(* IEC 61131-3 sources: volt/packages/volt-lsp-iec/test-corpus/lenze-mid/Device/Plc Logic/Application/Library Manager/L_MC4P_RoboticHandling, 315 files *)

(* ---- IDENT_IN_GROUP_REF.dut ---- *)
TYPE IDENT_IN_GROUP_REF :
(
	NONE := 0,
	X := 1,
	Y := 2,
	Z := 3,
	A := 4,
	B := 5,
	C := 6,
	A1 := 7,
	A2 := 8,
	A3 := 9,
	A4 := 10,
	A5 := 11,
	A6 := 12,
	AUX1 := 13,
	AUX2 := 14,
	AUX3 := 15,
	AUX4 := 16,
	AUX5 := 17,
	AUX6 := 18
);
END_TYPE

(* ---- L_MC4P_AGBC_PARAMETER.dut ---- *)
TYPE L_MC4P_AGBC_PARAMETER :
STRUCT
	LRCARTESIANJOGVEL : LREAL := 10;
	LRCARTESIANJOGACC : LREAL := 100;
	LRCARTESIANJOGDEC : LREAL := 200;
	LRCARTESIANJOGJERK : LREAL := 10000;
	LRORIENTATIONJOGVEL : LREAL := 5;
	LRORIENTATIONJOGACC : LREAL := 50;
	LRORIENTATIONJOGDEC : LREAL := 100;
	LRORIENTATIONJOGJERK : LREAL := 5000;
	LRREALAXISJOGVEL : LREAL := 5;
	LRREALAXISJOGACC : LREAL := 50;
	LRREALAXISJOGDEC : LREAL := 100;
	LRREALAXISJOGJERK : LREAL := 5000;
	LRCARTESIANMOVEVEL : LREAL := 10;
	LRCARTESIANMOVEACC : LREAL := 100;
	LRCARTESIANMOVEDEC : LREAL := 200;
	LRCARTESIANMOVEJERK : LREAL := 10000;
	LRORIENTATIONMOVEVEL : LREAL := 5;
	LRORIENTATIONMOVEACC : LREAL := 50;
	LRORIENTATIONMOVEDEC : LREAL := 100;
	LRORIENTATIONMOVEJERK : LREAL := 5000;
	LRREALAXISMOVEVEL : LREAL := 5;
	LRREALAXISMOVEACC : LREAL := 50;
	LRREALAXISMOVEDEC : LREAL := 100;
	LRREALAXISMOVEJERK : LREAL := 5000;
	LRPATHVEL : LREAL := 50;
	LRPATHACC : LREAL := 100;
	LRPATHDEC : LREAL := 100;
	LRPATHJERK : LREAL := 10000;
	LRPATHSTOPDEC : LREAL := 500;
	LRPATHSTOPJERK : LREAL := 50000;
	XGROUPSETPOSRELATIVE : BOOL := FALSE;
	ALRHOMEPOSITION : ARRAY [1..12] OF LREAL;
	AEHOMINGORDER : ARRAY [1..12] OF L_MC4P_HomingOrder;
	XUSEHOMEEXTPARAMETER : BOOL;
	ASCHOMEEXTPARAMETER : ARRAY [1..12] OF L_MC1P_HomeParameter;
	LRORFADINGTIME : LREAL := 2.5;
	EORIENTATIONMODE : L_MC4P_Orientation_Mode := L_MC4P_Orientation_Mode.ShortestSpacialWay;
	AEDIRECTION : ARRAY [1..6] OF MC_DIRECTION := [6(MC_DIRECTION.mcShortestWay)];
END_STRUCT
END_TYPE

(* ---- L_MC4P_AGBC_STATE.dut ---- *)
TYPE L_MC4P_AGBC_STATE :
(
	STANDBY := 0,
	STOP := 1,
	HOMING := 2,
	SETPOSITION := 3,
	MANMODE := 4,
	MOVELINABS := 5,
	MOVELINREL := 6,
	MOVEDIRABS := 7,
	MOVEDIRREL := 8,
	EXTERNAL := 9,
	SERVICE := 10,
	ERROR := 11,
	FINISHPOSITIONING := 12,
	PAUSE := 13
);
END_TYPE

(* ---- L_MC4P_ASCIIDECODERFILEDATA.dut ---- *)
TYPE L_MC4P_ASCIIDECODERFILEDATA :
STRUCT
	SFILENAME : STRING;
	IFILEID : INT;
	SPROGRAM : STRING;
	UDIPOS : UDINT;
	UDIPOSSTART : UDINT;
	UDIFILELENGTH : UDINT;
	LIFILELINENO : LINT;
	LISOURCELINENO : LINT;
	XLASTLINE : BOOL;
	XENDOFFILE : BOOL;
	XNEXTFILEVALID : BOOL;
	XDECODING : BOOL;
	XINIT : BOOL;
	XDONE : BOOL;
END_STRUCT
END_TYPE

(* ---- L_MC4P_ASCIIDECODERHEADDATA.dut ---- *)
TYPE L_MC4P_ASCIIDECODERHEADDATA :
STRUCT
	SCMODALDATA : L_MC4P_AsciiDecoderModalData;
	IACTIVEFILEID : INT := 1;
	ASCFILEDATA : ARRAY [1..GVL_MovePath.gciNumOfPathFiles] OF L_MC4P_AsciiDecoderFileData;
	SCTEMPDATA : L_MC4P_AsciiDecoderTempData;
	XADDPATHDATA : BOOL;
	XENDOFPROG : BOOL;
	XUPDATEFILE : BOOL;
	XWAITFORNEXTSOURCELINE : BOOL;
	XWAITFORBLOCKSEARCHLINE : BOOL;
	XINTERPRETERHALT : BOOL;
	XINTERPRETERHALTOLD : BOOL;
	BYADRESS : BYTE;
	STADRESSVALUE : STRING(255);
END_STRUCT
END_TYPE

(* ---- L_MC4P_ASCIIDECODERMODALDATA.dut ---- *)
TYPE L_MC4P_ASCIIDECODERMODALDATA :
STRUCT
	XRELATIVE : BOOL;
	XRELATIVEIJK : BOOL := TRUE;
	ECOORDSYSTEM : L_MC4P_CoordSystem := L_MC4P_CoordSystem.WCS;
	XCOORDSYSTEMVALID : BOOL;
	WCOORDLEVEL : WORD := 17;
	ALRNORMAL : ARRAY [1..3] OF LREAL := [0.0, 0.0, 1.0];
	ESEGMENTTYPE : L_MC4P_SegmentType;
	PATHCHOICE : MC_CIRC_PATHCHOICE;
	XSEGMENTTYPEVALID : BOOL;
	POSITION : ARRAY [1..12] OF LREAL;
	WPOSITIONMASK : WORD;
	LRPATHVEL : LREAL;
	LRPATHACC : LREAL;
	LRPATHDEC : LREAL;
	LRBLENDINGRADIUS : LREAL;
	XBLENDING : BOOL;
	LRBLENDINGRADIUS_OLD : LREAL;
	XBLENDING_OLD : BOOL;
	WPATHMASK : WORD;
END_STRUCT
END_TYPE

(* ---- L_MC4P_ASCIIDECODERTEMPDATA.dut ---- *)
TYPE L_MC4P_ASCIIDECODERTEMPDATA :
STRUCT
	LIN : LINT;
	XNVALID : BOOL;
	LRR : LREAL;
	XRVALID : BOOL;
	LRD : LREAL;
	XDVALID : BOOL;
	LRT : LREAL;
	XTVALID : BOOL;
	VECTOR : ARRAY [1..12] OF LREAL;
	WVECTORMASK : WORD;
	VECTORIJK : ARRAY [1..3] OF LREAL;
	WVECTORIJKMASK : WORD;
	XIJKASNORMAL : BOOL;
	ESEGMENTTYPE : L_MC4P_SegmentType;
	XG22 : BOOL;
	XLFILEVALID : BOOL;
	XGOTOACTIVE : BOOL;
	XIFACTIVE : BOOL;
	EGCODETYPE : L_MC4P_GCodeType;
	WMCOMMANDCOUNTER : WORD;
	EMFUNTYPE : L_MC4P_MFunctionType := L_MC4P_MFunctionType.inactive;
	LIMFUNID : LINT := 0;
	XHALTATSTART : BOOL;
	XHALTATEND : BOOL;
	AWMFUN : ARRAY [1..L_MC4P_Constants.gciMaxNumParallelMFun] OF WORD;
	SCPARAMSTORE : L_MC4P_MParams;
	WHCOMMANDCOUNTER : WORD;
	SCSWITCHINGFUN : L_MC4P_SwitchingFunctionData;
END_STRUCT
END_TYPE

(* ---- L_MC4P_AUXAXESDATA.dut ---- *)
TYPE L_MC4P_AUXAXESDATA :
STRUCT
	ALRAUXAXISTIMEOFFSET : ARRAY [1..6] OF LREAL;
	AXAUXAXISSEQACTIVE : ARRAY [1..6] OF BOOL;
	AXAUXAXISCALCPROFILE : ARRAY [1..6] OF BOOL;
	XAUXAXISCALCALLPROFILESNOW : BOOL;
	XAUXAXISACTIV : BOOL;
	ALRSTARTPOSAUX : ARRAY [1..6] OF LREAL;
	ALRTARGETPOSAUX : ARRAY [1..6] OF LREAL;
	AEAUXMODE : ARRAY [1..6] OF L_MC4P_AuxMode;
	ADIAUXAXISMODULOCOUTER : ARRAY [1..6] OF DINT;
END_STRUCT
END_TYPE

(* ---- L_MC4P_AUXMODE.dut ---- *)
TYPE L_MC4P_AUXMODE :
(
	INACTIVE := 0,
	CONTINUOUS := 1,
	DISCRETEABSOLUTE := 2,
	DISCRETERELATIVE := 3
);
END_TYPE

(* ---- L_MC4P_AXESGROUP_STATE.dut ---- *)
TYPE L_MC4P_AXESGROUP_STATE :
(
	GROUPERRORSTOP := 1,
	GROUPDISABLED := 2,
	GROUPSTANDBY := 3,
	GROUPSTOPPING := 4,
	GROUPMOVING := 5,
	GROUPHOMING := 6
);
END_TYPE

(* ---- L_MC4P_AXESGROUPMEMBER.dut ---- *)
TYPE L_MC4P_AXESGROUPMEMBER :
STRUCT
	LRMANUALMODETRANSVEL : LREAL;
	LRMANUALMODETRANSACC : LREAL;
	LRMANUALMODETRANSDEC : LREAL;
	LRMANUALMODETRANSJERK : LREAL;
	LRMANUALMODEROTVEL : LREAL;
	LRMANUALMODEROTACC : LREAL;
	LRMANUALMODEROTDEC : LREAL;
	LRMANUALMODEROTJERK : LREAL;
	LRPATHHALTDEC : LREAL;
	LRPATHHALTJERK : LREAL;
	AEHOMINGORDER : ARRAY [1..12] OF L_MC4P_HomingOrder;
END_STRUCT
END_TYPE

(* ---- L_MC4P_AXISENABLEMODE.dut ---- *)
TYPE L_MC4P_AXISENABLEMODE :
(
	DISABLE := 0,
	ENABLEPOSNEG := 1,
	ENABLEPOS := 2,
	ENABLENEG := 3
);
END_TYPE

(* ---- L_MC4P_AXISPROFILE.dut ---- *)
TYPE L_MC4P_AXISPROFILE :
STRUCT
	LRPOS : LREAL;
	LRVEL : LREAL;
	LRACC : LREAL;
END_STRUCT
END_TYPE

(* ---- L_MC4P_AXISTYPE.dut ---- *)
TYPE L_MC4P_AXISTYPE :
(
	UNCONNECTED := 0,
	LINEAR := 1,
	ROTARY := 2
);
END_TYPE

(* ---- L_MC4P_BLENDINGDATA.dut ---- *)
TYPE L_MC4P_BLENDINGDATA :
STRUCT
	LRLENGTHBLENDSTART : LREAL;
	LRLENGTHBLENDEND : LREAL;
	LRLENGTHNORMSTART : LREAL;
	LRLENGTHNORMEND : LREAL;
END_STRUCT
END_TYPE

(* ---- L_MC4P_CIRCLEDATA.dut ---- *)
TYPE L_MC4P_CIRCLEDATA :
STRUCT
	RESERVED : ARRAY [1..SIZEOF(L_MC4P_PathData)] OF BYTE;
	ALRCENTERPOINT : ARRAY [1..3] OF LREAL;
	LAMBDA_MAX : LREAL;
	ORIGIN_LAMBDA_MAX : LREAL;
	R_S : ARRAY [1..3, 1..3] OF LREAL;
	PATHCHOICE : MC_CIRC_PATHCHOICE;
	RADIUS : LREAL;
END_STRUCT
END_TYPE

(* ---- L_MC4P_CIRCMODE.dut ---- *)
TYPE L_MC4P_CIRCMODE :
(
	BORDER := 0,
	CENTER := 1,
	RADIUS := 2
);
END_TYPE

(* ---- L_MC4P_CLASSID.dut ---- *)
TYPE L_MC4P_CLASSID :
(
	AXES_GROUP_KIN := (L_MC4P_Internal.cdiEnumStartValue + 1),
	GROUPSTOP := (L_MC4P_Internal.cdiEnumStartValue + 4),
	GROUPHOME := (L_MC4P_Internal.cdiEnumStartValue + 5),
	GROUPMANUALMODE := (L_MC4P_Internal.cdiEnumStartValue + 6),
	GROUPSETOVERRIDE := (L_MC4P_Internal.cdiEnumStartValue + 7),
	GROUPREADSTATUS := (L_MC4P_Internal.cdiEnumStartValue + 8),
	GROUPSETPOSITION := (L_MC4P_Internal.cdiEnumStartValue + 9),
	GROUPRESET := (L_MC4P_Internal.cdiEnumStartValue + 10),
	GROUPENABLE := (L_MC4P_Internal.cdiEnumStartValue + 11),
	GROUPREADACTUALPOSITION := (L_MC4P_Internal.cdiEnumStartValue + 12),
	GROUPREADACTUALVELOCITY := (L_MC4P_Internal.cdiEnumStartValue + 13),
	GROUPWAITTIME := (L_MC4P_Internal.cdiEnumStartValue + 14),
	MC4P_FB_MOVECONTPATH := (L_MC4P_Internal.cdiEnumStartValue + 30),
	MC4P_FB_MOVELINEARABSOLUTE := (L_MC4P_Internal.cdiEnumStartValue + 31),
	MC4P_FB_MOVELINEARRELATIVE := (L_MC4P_Internal.cdiEnumStartValue + 32),
	MC4P_FB_MOVECIRCULARABSOLUTE := (L_MC4P_Internal.cdiEnumStartValue + 33),
	MC4P_FB_MOVECIRCULARRELATIVE := (L_MC4P_Internal.cdiEnumStartValue + 34),
	MC4P_FB_MOVEDIRECTRELATIVE := (L_MC4P_Internal.cdiEnumStartValue + 35),
	MC4P_FB_MOVEDIRECTABSOLUTE := (L_MC4P_Internal.cdiEnumStartValue + 36),
	MC4P_FB_MOVEELLIPTICALABSOLUTE := (L_MC4P_Internal.cdiEnumStartValue + 37),
	MC4P_FB_MOVEELLIPTICALRELATIVE := (L_MC4P_Internal.cdiEnumStartValue + 38),
	MC4P_FB_MOVEELLIPTICALPNP := (L_MC4P_Internal.cdiEnumStartValue + 39),
	MC4P_FB_MOVESPLINEABSOLUTE := (L_MC4P_Internal.cdiEnumStartValue + 40),
	MC4P_FB_MOVESPLINERELATIVE := (L_MC4P_Internal.cdiEnumStartValue + 41),
	MC4P_FB_MOVESPLINEPNP := (L_MC4P_Internal.cdiEnumStartValue + 42)
);
END_TYPE

(* ---- L_MC4P_COORDSYSTEM.dut ---- *)
TYPE L_MC4P_COORDSYSTEM :
(
	ACS := -1,
	WCS := 0,
	PCS_1 := 1,
	PCS_2 := 2,
	PCS_3 := 3,
	PCS_4 := 4,
	PCS_5 := 5,
	PCS_6 := 6,
	PCS_7 := 7,
	PCS_8 := 8,
	PCS_9 := 9,
	PCS_10 := 10,
	PCS_11 := 11,
	PCS_12 := 12,
	PCS_13 := 13,
	PCS_14 := 14,
	PCS_15 := 15,
	PCS_16 := 16,
	MCS := 1000
);
END_TYPE

(* ---- L_MC4P_COORDTYPE.dut ---- *)
TYPE L_MC4P_COORDTYPE :
(
	CARTESIAN := 0,
	CYLINDRIC := 1
);
END_TYPE

(* ---- L_MC4P_CUBICSPLINEDATA.dut ---- *)
TYPE L_MC4P_CUBICSPLINEDATA :
STRUCT
	RESERVED : ARRAY [1..SIZEOF(L_MC4P_PathData)] OF BYTE;
	ASCSPLINEDATA : ARRAY [1..10] OF L_MC4P_SplineData;
	UICNTINTERMEDIATEPOINTS : UINT;
	UIORIGINCNTINTERMEDIATEPOINTS : UINT;
END_STRUCT
END_TYPE

(* ---- L_MC4P_CYCLICDATA.dut ---- *)
TYPE L_MC4P_CYCLICDATA :
STRUCT
	LRT_ACT : LREAL := 0.001;
	ALRTAUX_ACT : ARRAY [1..6] OF LREAL;
	S_NORM : LREAL;
	DIGEOSEGMENTNO : DINT;
	DITIMESEGMENTNO : DINT;
	DISEGMENTNO : DINT;
	ETIMESEGMENTTYPE : L_MC4P_SegmentType;
	X_WCS : ARRAY [1..6] OF LREAL;
	V_WCS : ARRAY [1..6] OF LREAL;
	A_WCS : ARRAY [1..6] OF LREAL;
	X_WCSUNFILT : ARRAY [4..6] OF LREAL;
	V_WCSUNFILT : ARRAY [4..6] OF LREAL;
	A_WCSUNFILT : ARRAY [4..6] OF LREAL;
	ALRTANGENT : ARRAY [1..3] OF LREAL;
	ALRNORMAL : ARRAY [1..3] OF LREAL;
	ALRBINORMAL : ARRAY [1..3] OF LREAL;
	LRCURV : LREAL;
	X_AUX : ARRAY [1..6] OF LREAL;
	V_AUX : ARRAY [1..6] OF LREAL;
	A_AUX : ARRAY [1..6] OF LREAL;
	X_AUXUNFILT : ARRAY [1..6] OF LREAL;
	V_AUXUNFILT : ARRAY [1..6] OF LREAL;
	A_AUXUNFILT : ARRAY [1..6] OF LREAL;
	ADIAUXAXISMODULOCOUTER : ARRAY [1..6] OF DINT;
	X_ACS : ARRAY [1..6] OF LREAL;
	V_ACS : ARRAY [1..6] OF LREAL;
	A_ACS : ARRAY [1..6] OF LREAL;
	LRSETORIVEL : LREAL;
	LRSETORIACC : LREAL;
	LRSETPATHPOS : LREAL;
	LRSETPATHVEL : LREAL;
	LRSETPATHACC : LREAL;
	LRPASSEDLENGTHTIMESEGMENT : LREAL;
	LRPASSEDLENGTHGEOSEGMENT : LREAL;
	LRSETPATHPOSUNFILT : LREAL;
	LRSETPATHVELUNFILT : LREAL;
	LRSETPATHACCUNFILT : LREAL;
END_STRUCT
END_TYPE

(* ---- L_MC4P_DIFFGEARFACTORS2X2.dut ---- *)
TYPE L_MC4P_DIFFGEARFACTORS2X2 :
STRUCT
	DINUM12 : DINT;
	UDIDENUM12 : UDINT;
	DINUM21 : DINT;
	UDIDENUM21 : UDINT;
END_STRUCT
END_TYPE

(* ---- L_MC4P_DIFFGEARFACTORS3X3.dut ---- *)
TYPE L_MC4P_DIFFGEARFACTORS3X3 :
STRUCT
	DINUM12 : DINT;
	UDIDENUM12 : UDINT;
	DINUM13 : DINT;
	UDIDENUM13 : UDINT;
	DINUM23 : DINT;
	UDIDENUM23 : UDINT;
	DINUM21 : DINT;
	UDIDENUM21 : UDINT;
	DINUM31 : DINT;
	UDIDENUM31 : UDINT;
	DINUM32 : DINT;
	UDIDENUM32 : UDINT;
END_STRUCT
END_TYPE

(* ---- L_MC4P_ELLIPSEDATA.dut ---- *)
TYPE L_MC4P_ELLIPSEDATA :
STRUCT
	RESERVED : ARRAY [1..SIZEOF(L_MC4P_PathData)] OF BYTE;
	ALRCENTERPOINT : ARRAY [1..3] OF LREAL;
	LAMBDA_MAX : LREAL;
	ORIGIN_LAMBDA_MAX : LREAL;
	R_S : ARRAY [1..3, 1..3] OF LREAL;
	ORIGIN_R_S : ARRAY [1..3, 1..3] OF LREAL;
	PATHCHOICE : MC_CIRC_PATHCHOICE;
	ALR_RN_CIRC : ARRAY [1..3] OF LREAL;
	LRSEMIMAJORAXIS : LREAL;
	LRSEMIMINORAXIS : LREAL;
	LRECCENTRICITY : LREAL;
	LRPHI0 : LREAL;
	LRPHI1 : LREAL;
	LRORIGIN_PHI0 : LREAL;
	LRORIGIN_PHI1 : LREAL;
	LRARCLENGTH0 : LREAL;
END_STRUCT
END_TYPE

(* ---- L_MC4P_ELLIPTICALPNPMODE.dut ---- *)
TYPE L_MC4P_ELLIPTICALPNPMODE :
(
	ELLIPTICAL_180 := 1,
	ELLIPTICAL_90_STARTDIRECTION := 2,
	ELLIPTICAL_90_ENDDIRECTION := 3
);
END_TYPE

(* ---- L_MC4P_ERRORSTOPBEHAVIOUR.dut ---- *)
TYPE L_MC4P_ERRORSTOPBEHAVIOUR :
(
	SETTORQUETOZERO := 0,
	FADETORQUETOZERO := 1,
	CONTINUEPRECONTROL := 10
);
END_TYPE

(* ---- L_MC4P_ERRORSTRUCT.dut ---- *)
TYPE L_MC4P_ERRORSTRUCT :
STRUCT
	EERRORID : L_IE1P_Error;
	DWINTERNAL : DWORD;
END_STRUCT
END_TYPE

(* ---- L_MC4P_GCODETYPE.dut ---- *)
TYPE L_MC4P_GCODETYPE :
(
	UNDEFINED := 65535,
	G00 := 0,
	G01 := 1,
	G02 := 2,
	G03 := 3,
	G04 := 4,
	G16 := 16,
	G17 := 17,
	G18 := 18,
	G19 := 19,
	G22 := 22,
	G50 := 50,
	G51 := 51,
	G53 := 53,
	G54 := 54,
	G55 := 55,
	G56 := 56,
	G57 := 57,
	G58 := 58,
	G59 := 59,
	G75 := 75,
	G90 := 90,
	G91 := 91,
	G98 := 98,
	G99 := 99,
	ENDOFSUBROUTINE := 65029,
	ENDOFPROGRAM := 65030,
	MOS := 65100,
	MVS_SVS := 65200,
	MVS_SNS := 65300,
	MNS_SNS := 65400
);
END_TYPE

(* ---- L_MC4P_GEOOBJECTDATAUNION.dut ---- *)
TYPE L_MC4P_GEOOBJECTDATAUNION :
UNION
	AUXAXES : L_MC4P_AuxAxesData;
	PATH : L_MC4P_PathData;
	POLYNOM : L_MC4P_PolynomData;
	CIRCLE : L_MC4P_CircleData;
	CUBICSPLINE : L_MC4P_CubicSplineData;
	ELLIPSE : L_MC4P_EllipseData;
	PTP : L_MC4P_PTPData;
	WAITTIME : L_MC4P_WaitTimeData;
END_UNION
END_TYPE

(* ---- L_MC4P_GEOOBJECTINST.dut ---- *)
TYPE L_MC4P_GEOOBJECTINST :
STRUCT
	FBS2UMAP : L_UMTP_InterpolationLinear;
	SCS2UMAPDATA : L_UMTP_InterpolationData;
	XHASNONLINEARMAP : BOOL;
	ALR_U : ARRAY [1..2] OF LREAL;
	ALRLENGTH : ARRAY [1..L_MC4P_Constants.LengthVec_idxmax] OF LREAL;
END_STRUCT
END_TYPE

(* ---- L_MC4P_GROUPMANUALMODE_PARAMETER.dut ---- *)
TYPE L_MC4P_GROUPMANUALMODE_PARAMETER :
STRUCT
	LRCARTESIANJOGVEL : LREAL := 10;
	LRCARTESIANJOGACC : LREAL := 100;
	LRCARTESIANJOGDEC : LREAL := 200;
	LRCARTESIANJOGJERK : LREAL := 10000;
	LRORIENTATIONJOGVEL : LREAL := 5;
	LRORIENTATIONJOGACC : LREAL := 50;
	LRORIENTATIONJOGDEC : LREAL := 100;
	LRORIENTATIONJOGJERK : LREAL := 5000;
	LRREALAXISJOGVEL : LREAL := 5;
	LRREALAXISJOGACC : LREAL := 50;
	LRREALAXISJOGDEC : LREAL := 100;
	LRREALAXISJOGJERK : LREAL := 5000;
	LRCARTESIANMOVEVEL : LREAL := 10;
	LRCARTESIANMOVEACC : LREAL := 100;
	LRCARTESIANMOVEDEC : LREAL := 200;
	LRCARTESIANMOVEJERK : LREAL := 10000;
	LRORIENTATIONMOVEVEL : LREAL := 5;
	LRORIENTATIONMOVEACC : LREAL := 50;
	LRORIENTATIONMOVEDEC : LREAL := 100;
	LRORIENTATIONMOVEJERK : LREAL := 5000;
	LRREALAXISMOVEVEL : LREAL := 5;
	LRREALAXISMOVEACC : LREAL := 50;
	LRREALAXISMOVEDEC : LREAL := 100;
	LRREALAXISMOVEJERK : LREAL := 5000;
END_STRUCT
END_TYPE

(* ---- L_MC4P_HOMINGORDER.dut ---- *)
TYPE L_MC4P_HOMINGORDER :
(
	NOHOMING := 0,
	FIRST := 1,
	SECOND := 2,
	THIRD := 3,
	FOURTH := 4,
	FIFTH := 5,
	SIXTH := 6,
	SEVENTH := 7,
	EIGHTH := 8,
	NINTH := 9,
	TENTH := 10,
	ELEVENTH := 11,
	TWELFTH := 12
);
END_TYPE

(* ---- L_MC4P_IDENTMODE.dut ---- *)
TYPE L_MC4P_IDENTMODE :
(
	COMPLETEMODEL := 0,
	FRICTIONONLY := 1,
	RIGIDBODYONLY := 2
);
END_TYPE

(* ---- L_MC4P_IDENTTRAJECTORYFOURIERPARAM.dut ---- *)
TYPE L_MC4P_IDENTTRAJECTORYFOURIERPARAM :
STRUCT
	USIORDER : USINT;
	LRPERIOD : LREAL;
	ALRFREQUENCY : ARRAY [1..L_MC4P_Constants.gcusiMaxFourierCoeffsIdent] OF LREAL;
	LRA0_EXCITATION : LREAL;
	ALRAMPSINE_EXCITATION : ARRAY [1..L_MC4P_Constants.gcusiMaxFourierCoeffsIdent] OF LREAL;
	ALRAMPCOSINE_EXCITATION : ARRAY [1..L_MC4P_Constants.gcusiMaxFourierCoeffsIdent] OF LREAL;
	LRA0_AXES : LREAL;
	ALRAMPSINE_AXES : ARRAY [1..L_MC4P_Constants.gcusiMaxFourierCoeffsIdent] OF LREAL;
	ALRAMPCOSINE_AXES : ARRAY [1..L_MC4P_Constants.gcusiMaxFourierCoeffsIdent] OF LREAL;
END_STRUCT
END_TYPE

(* ---- L_MC4P_INTERMEDIATEPOINTSPLINE.dut ---- *)
TYPE L_MC4P_INTERMEDIATEPOINTSPLINE :
STRUCT
	LRXPOS : LREAL;
	LRYPOS : LREAL;
	LRZPOS : LREAL;
	XUSEPOINT : BOOL;
END_STRUCT
END_TYPE

(* ---- L_MC4P_INTERMEDIATERESULTSTORE.dut ---- *)
TYPE L_MC4P_INTERMEDIATERESULTSTORE :
STRUCT
	PX_FCS : POINTER TO LREAL;
	PV_FCS : POINTER TO LREAL;
	PA_FCS : POINTER TO LREAL;
	NDIMFCS : UDINT;
	PX_JCS : POINTER TO LREAL;
	PV_JCS : POINTER TO LREAL;
	PA_JCS : POINTER TO LREAL;
	NDIMJCS : UDINT;
	XFCSISCOMPUTED : BOOL;
	XMCSISCOMPUTED : BOOL;
	XWCSISCOMPUTED : BOOL;
END_STRUCT
END_TYPE

(* ---- L_MC4P_KINEMATICTYPE.dut ---- *)
TYPE L_MC4P_KINEMATICTYPE :
(
	NOKINEMATIC := 0,
	DELTA3_3DOF := 2,
	PORTAL_3DOF := 3,
	SCARA_3DOF := 5,
	SCARA_4DOF := 6,
	DELTA2_2DOF := 7,
	BELTKINEMATIC_2DOF := 8,
	ARTICULATEDP_4DOF := 9,
	PORTAL_6DOF := 10,
	ARTICULATEDROBOT_6DOF := 11,
	LINEARDELTA3_3DOF := 12,
	DELTA3_5DOF := 13,
	PORTAL_4DOF := 14,
	GENERIC_4DOF := 15,
	LINEARDELTA3_4DOF := 16,
	DELTA3_4DOF := 17,
	TDELTA3_3DOF := 18,
	TDELTA3_4DOF := 19,
	TDELTA3_5DOF := 20,
	PORTALAB_5DOF := 21,
	PORTALAC_5DOF := 22,
	PORTALBC_5DOF := 23
);
END_TYPE

(* ---- L_MC4P_LA_SEGMENTTYPE.dut ---- *)
TYPE L_MC4P_LA_SEGMENTTYPE :
(
	LA_SEG_00 := 0,
	LA_SEG_1A := 1,
	LA_SEG_1B := 2,
	LA_SEG_1C := 3,
	LA_SEG_1D := 4,
	LA_SEG_2B := 5,
	LA_SEG_2C := 6,
	LA_SEG_D := 7
);
END_TYPE

(* ---- L_MC4P_LIMITSUSED.dut ---- *)
TYPE L_MC4P_LIMITSUSED :
(
	VEL_CARTAXISX := 16#1,
	VEL_CARTAXISY := 16#2,
	VEL_CARTAXISZ := 16#4,
	VEL_CARTAXISA := 16#8,
	VEL_CARTAXISB := 16#10,
	VEL_CARTAXISC := 16#20,
	ACC_CARTAXISX := 16#40,
	ACC_CARTAXISY := 16#80,
	ACC_CARTAXISZ := 16#100,
	ACC_CARTAXISA := 16#200,
	ACC_CARTAXISB := 16#400,
	ACC_CARTAXISC := 16#800,
	JERK_CARTAXISX := 16#1000,
	JERK_CARTAXISY := 16#2000,
	JERK_CARTAXISZ := 16#4000,
	JERK_CARTAXISA := 16#8000,
	JERK_CARTAXISB := 16#10000,
	JERK_CARTAXISC := 16#20000,
	VEL_AG := 16#40000,
	ACC_AG := 16#80000,
	JERK_AG := 16#100000,
	VEL_FB := 16#200000,
	ACC_FB := 16#400000,
	JERK_FB := 16#800000,
	VEL_CARTAXISX_FB := 16#1000000,
	VEL_CARTAXISY_FB := 16#2000000,
	VEL_CARTAXISZ_FB := 16#4000000,
	VEL_CARTAXISA_FB := 16#8000000,
	VEL_CARTAXISB_FB := 16#10000000,
	VEL_CARTAXISC_FB := 16#20000000,
	ACC_CARTAXISX_FB := 16#40000000,
	ACC_CARTAXISY_FB := 16#80000000,
	ACC_CARTAXISZ_FB := 16#100000000,
	ACC_CARTAXISA_FB := 16#200000000,
	ACC_CARTAXISB_FB := 16#400000000,
	ACC_CARTAXISC_FB := 16#800000000,
	JERK_CARTAXISX_FB := 16#1000000000,
	JERK_CARTAXISY_FB := 16#2000000000,
	JERK_CARTAXISZ_FB := 16#4000000000,
	JERK_CARTAXISA_FB := 16#8000000000,
	JERK_CARTAXISB_FB := 16#10000000000,
	JERK_CARTAXISC_FB := 16#20000000000,
	TORQUELIMIT_A1 := 16#40000000000,
	TORQUELIMIT_A2 := 16#80000000000,
	TORQUELIMIT_A3 := 16#100000000000,
	TORQUELIMIT_A4 := 16#200000000000,
	TORQUELIMIT_A5 := 16#400000000000,
	TORQUELIMIT_A6 := 16#800000000000,
	CURRENTLIMIT_A1 := 16#1000000000000,
	CURRENTLIMIT_A2 := 16#2000000000000,
	CURRENTLIMIT_A3 := 16#4000000000000,
	CURRENTLIMIT_A4 := 16#8000000000000,
	CURRENTLIMIT_A5 := 16#10000000000000,
	CURRENTLIMIT_A6 := 16#20000000000000,
	SPEEDCTRLLIMIT_A1 := 16#40000000000000,
	SPEEDCTRLLIMIT_A2 := 16#80000000000000,
	SPEEDCTRLLIMIT_A3 := 16#100000000000000,
	SPEEDCTRLLIMIT_A4 := 16#200000000000000,
	SPEEDCTRLLIMIT_A5 := 16#400000000000000,
	SPEEDCTRLLIMIT_A6 := 16#800000000000000,
	POSCTRLLIMIT_A1 := 16#1000000000000000,
	POSCTRLLIMIT_A2 := 16#2000000000000000,
	POSCTRLLIMIT_A3 := 16#4000000000000000,
	POSCTRLLIMIT_A4 := 16#8000000000000000
);
END_TYPE

(* ---- L_MC4P_LISTELEMENT.dut ---- *)
TYPE L_MC4P_LISTELEMENT :
STRUCT
	DISEGMENTNO : DINT;
	DISEGMENTNOCOPIEDFROM : DINT;
	XSEGMENTCOPIED : BOOL := FALSE;
	BNOTINUSE : BOOL;
	DWMASK : L_MC4P_ModulMask;
	PRIGHT : POINTER TO L_MC4P_ListElement;
	PLEFT : POINTER TO L_MC4P_ListElement;
	SCLISTELEMENTDATA : L_MC4P_ListElementData;
	FBPROVIDER : L_MC4P_GeoObjectProvider;
	PPARENT : POINTER TO L_MC4P_PathDataList;
END_STRUCT
END_TYPE

(* ---- L_MC4P_LISTELEMENTDATA.dut ---- *)
TYPE L_MC4P_LISTELEMENTDATA :
STRUCT
	IGEO : L_MC4P_IGeoObject;
	IRESETGEO : L_MC4P_IResetable;
	UGEODATA : L_MC4P_GeoObjectDataUnion;
	SCTRACKINGDATA : L_MC4P_TrackingData;
	PCORRESPONDINGFB : POINTER TO L_MC4P_MoveContPath;
	SFBINSTANCE : STRING;
	ESEGMENTTYPE : L_MC4P_SegmentType;
	IPOTIME : LREAL;
	ORIGIN_X0 : ARRAY [1..6] OF LREAL;
	ORIGIN_X1 : ARRAY [1..6] OF LREAL;
	ORIGIN_X0_PTP : ARRAY [1..6] OF LREAL;
	ORIGIN_X1_PTP : ARRAY [1..6] OF LREAL;
	X0 : ARRAY [1..6] OF LREAL;
	X1 : ARRAY [1..6] OF LREAL;
	X0_PTP : ARRAY [1..6] OF LREAL;
	X1_PTP : ARRAY [1..6] OF LREAL;
	X0STRICH : ARRAY [1..3] OF LREAL;
	X1STRICH : ARRAY [1..3] OF LREAL;
	X02STRICH : ARRAY [1..3] OF LREAL;
	X12STRICH : ARRAY [1..3] OF LREAL;
	X0TOOLCHANGEOFFSET : ARRAY [1..3] OF LREAL;
	LENGTH : LREAL;
	THETA : LREAL;
	ORIGIN_LENGTH : LREAL;
	ORIGIN_THETA : LREAL;
	MAXBEND : LREAL;
	ALRORIPATHABC : ARRAY [1..3] OF LREAL;
	ALRORIPATHABC_ORIGINAL : ARRAY [1..3] OF LREAL;
	SPROFILEPARAMETERSORIGINAL : L_MC4P_ListElementOriginalParameters_Profiles;
	SPROFILES : L_MC4P_ListElementDataProfiles;
	SMOOTHTOLPERC : LREAL;
	SMOOTHRADIUS : LREAL;
	ESMOOTHTYPE : L_MC4P_SegmentType;
	BUFFERMODE : MC_BUFFER_MODE;
	ELOOKAHEAD_SEGMENTTYPE : L_MC4P_LA_SegmentType;
	LRLOOKAHEAD_LENGTH_1C : LREAL;
	SCTRAFOINFO_START : L_MC4P_TrafoInfo;
	SCTRAFOINFO_FINAL : L_MC4P_TrafoInfo;
	EORIENTATIONMODE : L_MC4P_Orientation_Mode;
	AEDIRECTION : ARRAY [1..6] OF MC_DIRECTION;
	SCSWITCHINGFUN : L_MC4P_SwitchingFunctionData;
	WLISTELEMDATASTATUS : WORD;
END_STRUCT
END_TYPE

(* ---- L_MC4P_LISTELEMENTDATAPROFILES.dut ---- *)
TYPE L_MC4P_LISTELEMENTDATAPROFILES :
STRUCT
	LRIPOENDTIME : LREAL;
	LRREMAININGFILTERTIME : LREAL;
	UPROFILES : L_MC4P_ListElementDataProfilesUnion;
END_STRUCT
END_TYPE

(* ---- L_MC4P_LISTELEMENTDATAPROFILESCP.dut ---- *)
TYPE L_MC4P_LISTELEMENTDATAPROFILESCP :
STRUCT
	ASCDATAXYZ : L_MC1P_ProfileData;
	ASCPARXYZ : L_MC1P_ProfileParameter;
	ASCDATAABC : ARRAY [1..3] OF L_MC1P_ProfileData;
	ASCPARABC : ARRAY [1..3] OF L_MC1P_ProfileParameter;
	ASCDATAAUX : ARRAY [1..6] OF L_MC1P_ProfileData;
	ASCPARAUX : ARRAY [1..6] OF L_MC1P_ProfileParameter;
END_STRUCT
END_TYPE

(* ---- L_MC4P_LISTELEMENTDATAPROFILESPTP.dut ---- *)
TYPE L_MC4P_LISTELEMENTDATAPROFILESPTP :
STRUCT
	ASCDATAPTP : ARRAY [1..6] OF L_MC1P_ProfileData;
	ASCPARPTP : ARRAY [1..6] OF L_MC1P_ProfileParameter;
END_STRUCT
END_TYPE

(* ---- L_MC4P_LISTELEMENTDATAPROFILESUNION.dut ---- *)
TYPE L_MC4P_LISTELEMENTDATAPROFILESUNION :
UNION
	CPDATA : L_MC4P_ListElementDataProfilesCP;
	PTPDATA : L_MC4P_ListElementDataProfilesPTP;
END_UNION
END_TYPE

(* ---- L_MC4P_LISTELEMENTORIGINALPARAMETERS_PROFILES.dut ---- *)
TYPE L_MC4P_LISTELEMENTORIGINALPARAMETERS_PROFILES :
STRUCT
	LRVMAX : LREAL;
	LRAMAX : LREAL;
	LRDMAX : LREAL;
	LRJERK : LREAL;
	ALRJERKROT : ARRAY [1..3] OF LREAL;
	ALRVMAXROT : ARRAY [1..3] OF LREAL;
	ALRAMAXROT : ARRAY [1..3] OF LREAL;
END_STRUCT
END_TYPE

(* ---- L_MC4P_MANUALMODE.dut ---- *)
TYPE L_MC4P_MANUALMODE :
(
	STANDBY := 0,
	JOGGING := 1,
	MOVEREL := 2,
	MOVEABS := 3
);
END_TYPE

(* ---- L_MC4P_MAXVALUESOURCE.dut ---- *)
TYPE L_MC4P_MAXVALUESOURCE :
(
	AXISMAXORAPPLFB := 0,
	AXISDEFAULTORAPPLFB := 1,
	AXISDEFAULTORAPPLFBPRIODEFAULT := 2,
	AXISMAXORAPPLFBPRIOMAX := 3
);
END_TYPE

(* ---- L_MC4P_MEASUREDPROFILETIME.dut ---- *)
TYPE L_MC4P_MEASUREDPROFILETIME :
STRUCT
	WMASK : WORD;
	LRACTTIME : LREAL;
	LRPRECALTIME : LREAL;
END_STRUCT
END_TYPE

(* ---- L_MC4P_MFUNCTIONTYPE.dut ---- *)
TYPE L_MC4P_MFUNCTIONTYPE :
(
	INACTIVE := 0,
	MOS := 1,
	MVS_SVS := 2,
	MVS_SNS := 3,
	MNS_SNS := 4,
	NOTSUPPORTED := 100
);
END_TYPE

(* ---- L_MC4P_MODULMASK.dut ---- *)
TYPE L_MC4P_MODULMASK :
(
	L_MC4P_INITIAL_MASK := 16#0,
	L_MC4P_INTERPRETER_MASK := 16#1,
	L_MC4P_SMOOTHPATH_MASK := 16#3,
	L_MC4P_CALCULATEPATHPOLYNOM_MASK := 16#7,
	L_MC4P_CHECKWORKSPACE_MASK := 16#F,
	L_MC4P_LIMITDYNAMICSELEMENTS_MASK := 16#1F,
	L_MC4P_LIMITDYNAMICSCORNER_MASK := 16#3F,
	L_MC4P_LIMITDYNAMICSPATHLENGTH_MASK := 16#7F,
	L_MC4P_LIMITDYNAMICSCOMBINE_MASK := 16#FF,
	L_MC4P_CALCULATEPROFILEPOLYNOM_MASK := 16#1FF,
	L_MC4P_PREPAREAUXDATA_MASK := 16#3FF,
	L_MC4P_LA_CLEANUP_MASK := 16#7FF,
	L_MC4P_ACTIVATESEGMENT_MASK := 16#FFF,
	L_MC4P_TIMEINTERPOLATOR_MASK := 16#1FFF,
	L_MC4P_GEOINTERPOLATOR_MASK := 16#3FFF,
	L_MC4P_ELEMENT_BE_DELETED_MASK := 16#7FFF
);
END_TYPE

(* ---- L_MC4P_MOVECONTSTATES.dut ---- *)
TYPE L_MC4P_MOVECONTSTATES :
(
	INITIAL := 0,
	READPARAM_STANDBY := 100,
	READ_INPUTS := 1000,
	CALCPATH := 1100,
	IPO_STANDBY := 2000,
	IPO_ACTIVE := 2100,
	ABORTING := 8888,
	ERRORSTATE := 9999
);
END_TYPE

(* ---- L_MC4P_MOVEPATHSTORE.dut ---- *)
TYPE L_MC4P_MOVEPATHSTORE :
STRUCT
	FB_SEMAMOVEPATHFBS : L_MC1P_CriticalSection;
	AMOVECONTPATH : ARRAY [1..L_MC4P_Constants.ciNumOfMoveContPath] OF L_MC4P_MoveContPath;
END_STRUCT
END_TYPE

(* ---- L_MC4P_MPARAMS.dut ---- *)
TYPE L_MC4P_MPARAMS :
STRUCT
	LRPA : LREAL;
	LRPB : LREAL;
	LRPC : LREAL;
	LRPD : LREAL;
	LRPE : LREAL;
	LRPF : LREAL;
	LRPG : LREAL;
	LRPH : LREAL;
	LRPI : LREAL;
	LRPJ : LREAL;
	LRPK : LREAL;
	LRPL : LREAL;
	LRPM : LREAL;
	LRPN : LREAL;
	LRPO : LREAL;
	LRPP : LREAL;
	LRPQ : LREAL;
	LRPR : LREAL;
	LRPS : LREAL;
	LRPT : LREAL;
	LRPU : LREAL;
	LRPV : LREAL;
	LRPW : LREAL;
	LRPX : LREAL;
	LRPY : LREAL;
	LRPZ : LREAL;
END_STRUCT
END_TYPE

(* ---- L_MC4P_OBSERVATIONMODE.dut ---- *)
TYPE L_MC4P_OBSERVATIONMODE :
(
	FORCE := 1,
	MASS := 2
);
END_TYPE

(* ---- L_MC4P_ORIENTATION_MODE.dut ---- *)
TYPE L_MC4P_ORIENTATION_MODE :
(
	SHORTESTSPACIALWAY := 0,
	AXISINDIVIDUAL := 10
);
END_TYPE

(* ---- L_MC4P_OVRTYPE.dut ---- *)
TYPE L_MC4P_OVRTYPE :
(
	OVRTYPEPOLY := 1,
	OVRTYPEFAST := 2,
	OVRTYPECOMBINED := 3,
	OVRTYPEPT2 := 4
);
END_TYPE

(* ---- L_MC4P_PARACCESS.dut ---- *)
TYPE L_MC4P_PARACCESS :
STRUCT
	AXESGROUPNAME : REFERENCE TO STRING;
	KINEMATICTYPE : REFERENCE TO WORD;
	AXESGROUPSTATE : REFERENCE TO WORD;
	AXESGROUPSTATUSWORD : REFERENCE TO DWORD;
	ACTIVEERRORID : REFERENCE TO WORD;
	PATHSETVELOCITY : REFERENCE TO LREAL;
	PATHSETACCELERATION : REFERENCE TO LREAL;
	USEREALDRIVESASVIRTUAL : REFERENCE TO BOOL;
	HORIZONOFPATHPLANNING : REFERENCE TO WORD;
	DEFAULTORIENTATIONVELOCITY : REFERENCE TO LREAL;
	DEFAULTORIENTATIONACCELERATION : REFERENCE TO LREAL;
	DEFAULTORIENTATIONJERK : REFERENCE TO LREAL;
	TASKLOADPATHPREPERATION : REFERENCE TO WORD;
	ENABLEFULLBLENDING : REFERENCE TO BOOL;
	LIMITATIONOFPATH : REFERENCE TO WORD;
	ANGULARTOLERANCEEXACTSTOP : REFERENCE TO LREAL;
	MAXACCELERATIONDIFFERENCE : REFERENCE TO LREAL;
	ROTATIONCONVENTION : REFERENCE TO WORD;
	LIMITPATHTOMAINAXES : REFERENCE TO BOOL;
	JERKLIMITATION : REFERENCE TO WORD;
	SRAMPTIME : REFERENCE TO UINT;
	MAXPATHVELOCITY : REFERENCE TO LREAL;
	MAXPATHACCELERATION : REFERENCE TO LREAL;
	MAXPATHJERK : REFERENCE TO LREAL;
	HOMINGORDERA1 : REFERENCE TO WORD;
	HOMINGORDERA2 : REFERENCE TO WORD;
	HOMINGORDERA3 : REFERENCE TO WORD;
	HOMINGORDERA4 : REFERENCE TO WORD;
	HOMINGORDERA5 : REFERENCE TO WORD;
	HOMINGORDERA6 : REFERENCE TO WORD;
	HOMINGORDERAUX1 : REFERENCE TO WORD;
	HOMINGORDERAUX2 : REFERENCE TO WORD;
	HOMINGORDERAUX3 : REFERENCE TO WORD;
	HOMINGORDERAUX4 : REFERENCE TO WORD;
	HOMINGORDERAUX5 : REFERENCE TO WORD;
	HOMINGORDERAUX6 : REFERENCE TO WORD;
	REAKTONMCFBERROR : REFERENCE TO BOOL;
	ENABLELOGENTRY : REFERENCE TO BOOL;
	MANUALMODETRANSVEL : REFERENCE TO LREAL;
	MANUALMODETRANSACC : REFERENCE TO LREAL;
	MANUELMODETRANSDEC : REFERENCE TO LREAL;
	MANUALMODETRANSJERK : REFERENCE TO LREAL;
	MANUALMODEROTVEL : REFERENCE TO LREAL;
	MANUALMODEROTACC : REFERENCE TO LREAL;
	MANUALMODEROTDEC : REFERENCE TO LREAL;
	MANUALMODEROTJERK : REFERENCE TO LREAL;
	PATHHALTDEC : REFERENCE TO LREAL;
	PATHHALTJERK : REFERENCE TO LREAL;
	PCS_1_COORDTYPE : REFERENCE TO WORD;
	PCS_1_X : REFERENCE TO LREAL;
	PCS_1_Y : REFERENCE TO LREAL;
	PCS_1_Z : REFERENCE TO LREAL;
	PCS_1_A : REFERENCE TO LREAL;
	PCS_1_B : REFERENCE TO LREAL;
	PCS_1_C : REFERENCE TO LREAL;
	PCS_2_COORDTYPE : REFERENCE TO WORD;
	PCS_2_X : REFERENCE TO LREAL;
	PCS_2_Y : REFERENCE TO LREAL;
	PCS_2_Z : REFERENCE TO LREAL;
	PCS_2_A : REFERENCE TO LREAL;
	PCS_2_B : REFERENCE TO LREAL;
	PCS_2_C : REFERENCE TO LREAL;
	PCS_3_COORDTYPE : REFERENCE TO WORD;
	PCS_3_X : REFERENCE TO LREAL;
	PCS_3_Y : REFERENCE TO LREAL;
	PCS_3_Z : REFERENCE TO LREAL;
	PCS_3_A : REFERENCE TO LREAL;
	PCS_3_B : REFERENCE TO LREAL;
	PCS_3_C : REFERENCE TO LREAL;
	PCS_4_COORDTYPE : REFERENCE TO WORD;
	PCS_4_X : REFERENCE TO LREAL;
	PCS_4_Y : REFERENCE TO LREAL;
	PCS_4_Z : REFERENCE TO LREAL;
	PCS_4_A : REFERENCE TO LREAL;
	PCS_4_B : REFERENCE TO LREAL;
	PCS_4_C : REFERENCE TO LREAL;
	PCS_5_COORDTYPE : REFERENCE TO WORD;
	PCS_5_X : REFERENCE TO LREAL;
	PCS_5_Y : REFERENCE TO LREAL;
	PCS_5_Z : REFERENCE TO LREAL;
	PCS_5_A : REFERENCE TO LREAL;
	PCS_5_B : REFERENCE TO LREAL;
	PCS_5_C : REFERENCE TO LREAL;
	PCS_6_COORDTYPE : REFERENCE TO WORD;
	PCS_6_X : REFERENCE TO LREAL;
	PCS_6_Y : REFERENCE TO LREAL;
	PCS_6_Z : REFERENCE TO LREAL;
	PCS_6_A : REFERENCE TO LREAL;
	PCS_6_B : REFERENCE TO LREAL;
	PCS_6_C : REFERENCE TO LREAL;
	PCS_7_COORDTYPE : REFERENCE TO WORD;
	PCS_7_X : REFERENCE TO LREAL;
	PCS_7_Y : REFERENCE TO LREAL;
	PCS_7_Z : REFERENCE TO LREAL;
	PCS_7_A : REFERENCE TO LREAL;
	PCS_7_B : REFERENCE TO LREAL;
	PCS_7_C : REFERENCE TO LREAL;
	PCS_8_COORDTYPE : REFERENCE TO WORD;
	PCS_8_X : REFERENCE TO LREAL;
	PCS_8_Y : REFERENCE TO LREAL;
	PCS_8_Z : REFERENCE TO LREAL;
	PCS_8_A : REFERENCE TO LREAL;
	PCS_8_B : REFERENCE TO LREAL;
	PCS_8_C : REFERENCE TO LREAL;
	PCS_9_COORDTYPE : REFERENCE TO WORD;
	PCS_9_X : REFERENCE TO LREAL;
	PCS_9_Y : REFERENCE TO LREAL;
	PCS_9_Z : REFERENCE TO LREAL;
	PCS_9_A : REFERENCE TO LREAL;
	PCS_9_B : REFERENCE TO LREAL;
	PCS_9_C : REFERENCE TO LREAL;
	PCS_10_COORDTYPE : REFERENCE TO WORD;
	PCS_10_X : REFERENCE TO LREAL;
	PCS_10_Y : REFERENCE TO LREAL;
	PCS_10_Z : REFERENCE TO LREAL;
	PCS_10_A : REFERENCE TO LREAL;
	PCS_10_B : REFERENCE TO LREAL;
	PCS_10_C : REFERENCE TO LREAL;
	PCS_11_COORDTYPE : REFERENCE TO WORD;
	PCS_11_X : REFERENCE TO LREAL;
	PCS_11_Y : REFERENCE TO LREAL;
	PCS_11_Z : REFERENCE TO LREAL;
	PCS_11_A : REFERENCE TO LREAL;
	PCS_11_B : REFERENCE TO LREAL;
	PCS_11_C : REFERENCE TO LREAL;
	PCS_12_COORDTYPE : REFERENCE TO WORD;
	PCS_12_X : REFERENCE TO LREAL;
	PCS_12_Y : REFERENCE TO LREAL;
	PCS_12_Z : REFERENCE TO LREAL;
	PCS_12_A : REFERENCE TO LREAL;
	PCS_12_B : REFERENCE TO LREAL;
	PCS_12_C : REFERENCE TO LREAL;
	PCS_13_COORDTYPE : REFERENCE TO WORD;
	PCS_13_X : REFERENCE TO LREAL;
	PCS_13_Y : REFERENCE TO LREAL;
	PCS_13_Z : REFERENCE TO LREAL;
	PCS_13_A : REFERENCE TO LREAL;
	PCS_13_B : REFERENCE TO LREAL;
	PCS_13_C : REFERENCE TO LREAL;
	PCS_14_COORDTYPE : REFERENCE TO WORD;
	PCS_14_X : REFERENCE TO LREAL;
	PCS_14_Y : REFERENCE TO LREAL;
	PCS_14_Z : REFERENCE TO LREAL;
	PCS_14_A : REFERENCE TO LREAL;
	PCS_14_B : REFERENCE TO LREAL;
	PCS_14_C : REFERENCE TO LREAL;
	PCS_15_COORDTYPE : REFERENCE TO WORD;
	PCS_15_X : REFERENCE TO LREAL;
	PCS_15_Y : REFERENCE TO LREAL;
	PCS_15_Z : REFERENCE TO LREAL;
	PCS_15_A : REFERENCE TO LREAL;
	PCS_15_B : REFERENCE TO LREAL;
	PCS_15_C : REFERENCE TO LREAL;
	PCS_16_COORDTYPE : REFERENCE TO WORD;
	PCS_16_X : REFERENCE TO LREAL;
	PCS_16_Y : REFERENCE TO LREAL;
	PCS_16_Z : REFERENCE TO LREAL;
	PCS_16_A : REFERENCE TO LREAL;
	PCS_16_B : REFERENCE TO LREAL;
	PCS_16_C : REFERENCE TO LREAL;
	MCS_X : REFERENCE TO LREAL;
	MCS_Y : REFERENCE TO LREAL;
	MCS_Z : REFERENCE TO LREAL;
	MCS_A : REFERENCE TO LREAL;
	MCS_B : REFERENCE TO LREAL;
	MCS_C : REFERENCE TO LREAL;
	ACTIVETOOL : REFERENCE TO WORD;
	TOOL_1_TOOLTYPE : REFERENCE TO WORD;
	TOOL_1_X : REFERENCE TO LREAL;
	TOOL_1_Y : REFERENCE TO LREAL;
	TOOL_1_Z : REFERENCE TO LREAL;
	TOOL_1_A : REFERENCE TO LREAL;
	TOOL_1_B : REFERENCE TO LREAL;
	TOOL_1_C : REFERENCE TO LREAL;
	TOOL_1_SWITCHONTIME : REFERENCE TO INT;
	TOOL_1_SWITCHOFFTIME : REFERENCE TO INT;
	TOOL_2_TOOLTYPE : REFERENCE TO WORD;
	TOOL_2_X : REFERENCE TO LREAL;
	TOOL_2_Y : REFERENCE TO LREAL;
	TOOL_2_Z : REFERENCE TO LREAL;
	TOOL_2_A : REFERENCE TO LREAL;
	TOOL_2_B : REFERENCE TO LREAL;
	TOOL_2_C : REFERENCE TO LREAL;
	TOOL_2_SWITCHONTIME : REFERENCE TO INT;
	TOOL_2_SWITCHOFFTIME : REFERENCE TO INT;
	TOOL_3_TOOLTYPE : REFERENCE TO WORD;
	TOOL_3_X : REFERENCE TO LREAL;
	TOOL_3_Y : REFERENCE TO LREAL;
	TOOL_3_Z : REFERENCE TO LREAL;
	TOOL_3_A : REFERENCE TO LREAL;
	TOOL_3_B : REFERENCE TO LREAL;
	TOOL_3_C : REFERENCE TO LREAL;
	TOOL_3_SWITCHONTIME : REFERENCE TO INT;
	TOOL_3_SWITCHOFFTIME : REFERENCE TO INT;
	TOOL_4_TOOLTYPE : REFERENCE TO WORD;
	TOOL_4_X : REFERENCE TO LREAL;
	TOOL_4_Y : REFERENCE TO LREAL;
	TOOL_4_Z : REFERENCE TO LREAL;
	TOOL_4_A : REFERENCE TO LREAL;
	TOOL_4_B : REFERENCE TO LREAL;
	TOOL_4_C : REFERENCE TO LREAL;
	TOOL_4_SWITCHONTIME : REFERENCE TO INT;
	TOOL_4_SWITCHOFFTIME : REFERENCE TO INT;
	COULOMBFRICTIONA1 : REFERENCE TO LREAL;
	COULOMBFRICTIONA2 : REFERENCE TO LREAL;
	COULOMBFRICTIONA3 : REFERENCE TO LREAL;
	COULOMBFRICTIONA4 : REFERENCE TO LREAL;
	COULOMBFRICTIONA5 : REFERENCE TO LREAL;
	COULOMBFRICTIONA6 : REFERENCE TO LREAL;
	VISCOSEFRICTIONA1 : REFERENCE TO LREAL;
	VISCOSEFRICTIONA2 : REFERENCE TO LREAL;
	VISCOSEFRICTIONA3 : REFERENCE TO LREAL;
	VISCOSEFRICTIONA4 : REFERENCE TO LREAL;
	VISCOSEFRICTIONA5 : REFERENCE TO LREAL;
	VISCOSEFRICTIONA6 : REFERENCE TO LREAL;
	GRAVITATIONX : REFERENCE TO LREAL;
	GRAVITATIONY : REFERENCE TO LREAL;
	GRAVITATIONZ : REFERENCE TO LREAL;
	MINIMALDYNAMICPARAMETER1 : REFERENCE TO LREAL;
	MINIMALDYNAMICPARAMETER2 : REFERENCE TO LREAL;
	MINIMALDYNAMICPARAMETER3 : REFERENCE TO LREAL;
	MINIMALDYNAMICPARAMETER4 : REFERENCE TO LREAL;
	MINIMALDYNAMICPARAMETER5 : REFERENCE TO LREAL;
	MINIMALDYNAMICPARAMETER6 : REFERENCE TO LREAL;
	MINIMALDYNAMICPARAMETER7 : REFERENCE TO LREAL;
	MINIMALDYNAMICPARAMETER8 : REFERENCE TO LREAL;
	MINIMALDYNAMICPARAMETER9 : REFERENCE TO LREAL;
	MINIMALDYNAMICPARAMETER10 : REFERENCE TO LREAL;
	MINIMALDYNAMICPARAMETER11 : REFERENCE TO LREAL;
	MINIMALDYNAMICPARAMETER12 : REFERENCE TO LREAL;
	MINIMALDYNAMICPARAMETER13 : REFERENCE TO LREAL;
	MINIMALDYNAMICPARAMETER14 : REFERENCE TO LREAL;
	MINIMALDYNAMICPARAMETER15 : REFERENCE TO LREAL;
	MINIMALDYNAMICPARAMETER16 : REFERENCE TO LREAL;
	MINIMALDYNAMICPARAMETER17 : REFERENCE TO LREAL;
	MINIMALDYNAMICPARAMETER18 : REFERENCE TO LREAL;
END_STRUCT
END_TYPE

(* ---- L_MC4P_PARAMETER_MCMOVE.dut ---- *)
TYPE L_MC4P_PARAMETER_MCMOVE :
STRUCT
	POSITION : ARRAY [1..12] OF LREAL;
	DISTANCE : ARRAY [1..12] OF LREAL;
	XMOVEREL : BOOL;
	CIRCMODE : L_MC4P_CircMode;
	AUXPOINT : ARRAY [1..12] OF LREAL;
	PATHCHOICE : MC_CIRC_PATHCHOICE;
	LRSEMIMAJORAXIS : LREAL;
	LRSEMIMINORAXIS : LREAL;
	EELLIPTICALPNPMODE : L_MC4P_EllipticalPnPMode;
	ASCINTERMEDIATEPOINTSPLINE : ARRAY [1..GVL_MoveSpline.maxIntermediatePoints] OF L_MC4P_IntermediatePointSpline;
	VELOCITY : LREAL;
	ACCELERATION : LREAL;
	DECELERATION : LREAL;
	JERK : LREAL;
	ALRVELOCITYPTP : ARRAY [1..6] OF LREAL;
	ALRACCELERATIONPTP : ARRAY [1..6] OF LREAL;
	ALRDECELERATIONPTP : ARRAY [1..6] OF LREAL;
	ALRJERKPTP : ARRAY [1..6] OF LREAL;
	ALRVELOCITYAUX : ARRAY [1..6] OF LREAL;
	ALRACCELERATIONAUX : ARRAY [1..6] OF LREAL;
	ALRDECELERATIONAUX : ARRAY [1..6] OF LREAL;
	ALRJERKAUX : ARRAY [1..6] OF LREAL;
	COORDSYSTEM : L_MC4P_CoordSystem;
	COORDREF : MC_COORD_REF;
	BUFFERMODE : MC_BUFFER_MODE;
	TRANSITIONMODE : MC_TRANSITION_MODE;
	TRANSITIONPARAMETER : ARRAY [1..12] OF LREAL;
	AEAUXMODE : ARRAY [1..6] OF L_MC4P_AuxMode;
	ETOOLSYSTEM : L_MC4P_ToolSystem;
	ALRAXISLIMITVEL : ARRAY [1..18] OF LREAL;
	ALRAXISLIMITACC : ARRAY [1..18] OF LREAL;
	ALRAXISLIMITJERK : ARRAY [1..18] OF LREAL;
	AITARGETCONFIGURATION : ARRAY [1..6] OF INT;
	XWTRACKINGINSTANCE : __XWORD;
	EORIENTATIONMODE : L_MC4P_Orientation_Mode;
	AEDIRECTION : ARRAY [1..6] OF MC_DIRECTION;
	DWMASKMOVEPATH : DWORD;
	DWMASKVALIDVALUES : DWORD;
	ESEGMENTTYPE : L_MC4P_SegmentType;
	ESEGMENTTYPENEXT : L_MC4P_SegmentType;
	XAUXPOINTRELATIVE : BOOL;
	LIFILELINENO : LINT;
	LISOURCELINE : LINT;
	STSOURCE : STRING(255);
	LRWAITTIME : LREAL;
	NORMVECTOROFCOORDLEVEL : ARRAY [1..3] OF LREAL;
	CIRCRADIUS : LREAL;
	LRTARGETPOSTOLERANCE : LREAL := L_UMTP_Math.EPS_REAL;
	AIMOVECONTPATHNO : ARRAY [1..2] OF INT;
	INUMOFCONTPATH : INT := 1;
	XDONTCALCPROFILEMOVEPATH : BOOL;
	LRESTIMATEDSEGMENTLENGTH : LREAL;
	LRESTIMATEDSEGMENTTIME : LREAL;
	LRZMAXHEIGHT : LREAL;
	LRZSTARTDIST : LREAL;
	LRZTARGETDIST : LREAL;
	EGCODETYPE : L_MC4P_GCodeType;
	AWMFUN : ARRAY [1..L_MC4P_Constants.gciMaxNumParallelMFun] OF WORD;
	SCPARAMSTORE : L_MC4P_MParams;
	EMFUNTYPE : L_MC4P_MFunctionType;
	WMFUNID : WORD;
	XHALTATSTART : BOOL;
	XHALTATEND : BOOL;
	SCSWITCHINGFUN : L_MC4P_SwitchingFunctionData;
END_STRUCT
END_TYPE

(* ---- L_MC4P_PARAMETERINDEX.dut ---- *)
TYPE L_MC4P_PARAMETERINDEX :
(
	ONEOFFOUR := 104,
	TWOOFFOUR := 204,
	THREEOFFOUR := 304,
	FOUROFFOUR := 404
);
END_TYPE

(* ---- L_MC4P_PARAMS.dut ---- *)
TYPE L_MC4P_PARAMS :
(
	AXESGROUPNAME := 2,
	KINEMATICTYPE := 3,
	AXESGROUPSTATE := 4,
	AXESGROUPSTATUSWORD := 5,
	ACTIVEERRORID := 6,
	PATHSETVELOCITY := 15,
	PATHSETACCELERATION := 16,
	USEREALDRIVESASVIRTUAL := 29,
	HORIZONOFPATHPLANNING := 30,
	DEFAULTORIENTATIONVELOCITY := 31,
	DEFAULTORIENTATIONACCELERATION := 32,
	DEFAULTORIENTATIONJERK := 33,
	TASKLOADPATHPREPERATION := 34,
	ENABLEFULLBLENDING := 35,
	LIMITATIONOFPATH := 36,
	ANGULARTOLERANCEEXACTSTOP := 37,
	MAXACCELERATIONDIFFERENCE := 38,
	ROTATIONCONVENTION := 39,
	LIMITPATHTOMAINAXES := 40,
	JERKLIMITATION := 41,
	SRAMPTIME := 42,
	MAXPATHVELOCITY := 45,
	MAXPATHACCELERATION := 46,
	MAXPATHJERK := 47,
	HOMINGORDERA1 := 70,
	HOMINGORDERA2 := 71,
	HOMINGORDERA3 := 72,
	HOMINGORDERA4 := 73,
	HOMINGORDERA5 := 74,
	HOMINGORDERA6 := 75,
	HOMINGORDERAUX1 := 76,
	HOMINGORDERAUX2 := 77,
	HOMINGORDERAUX3 := 78,
	HOMINGORDERAUX4 := 79,
	HOMINGORDERAUX5 := 80,
	HOMINGORDERAUX6 := 81,
	REAKTONMCFBERROR := 102,
	ENABLELOGENTRY := 103,
	MANUALMODETRANSVEL := 181,
	MANUALMODETRANSACC := 182,
	MANUELMODETRANSDEC := 183,
	MANUALMODETRANSJERK := 184,
	MANUALMODEROTVEL := 186,
	MANUALMODEROTACC := 187,
	MANUALMODEROTDEC := 188,
	MANUALMODEROTJERK := 189,
	PATHHALTDEC := 190,
	PATHHALTJERK := 191,
	PCS_1_COORDTYPE := 1002,
	PCS_1_X := 1003,
	PCS_1_Y := 1004,
	PCS_1_Z := 1005,
	PCS_1_A := 1006,
	PCS_1_B := 1007,
	PCS_1_C := 1008,
	PCS_2_COORDTYPE := 1009,
	PCS_2_X := 1010,
	PCS_2_Y := 1011,
	PCS_2_Z := 1012,
	PCS_2_A := 1013,
	PCS_2_B := 1014,
	PCS_2_C := 1015,
	PCS_3_COORDTYPE := 1016,
	PCS_3_X := 1017,
	PCS_3_Y := 1018,
	PCS_3_Z := 1019,
	PCS_3_A := 1020,
	PCS_3_B := 1021,
	PCS_3_C := 1022,
	PCS_4_COORDTYPE := 1023,
	PCS_4_X := 1024,
	PCS_4_Y := 1025,
	PCS_4_Z := 1026,
	PCS_4_A := 1027,
	PCS_4_B := 1028,
	PCS_4_C := 1029,
	PCS_5_COORDTYPE := 1030,
	PCS_5_X := 1031,
	PCS_5_Y := 1032,
	PCS_5_Z := 1033,
	PCS_5_A := 1034,
	PCS_5_B := 1035,
	PCS_5_C := 1036,
	PCS_6_COORDTYPE := 1037,
	PCS_6_X := 1038,
	PCS_6_Y := 1039,
	PCS_6_Z := 1040,
	PCS_6_A := 1041,
	PCS_6_B := 1042,
	PCS_6_C := 1043,
	PCS_7_COORDTYPE := 1044,
	PCS_7_X := 1045,
	PCS_7_Y := 1046,
	PCS_7_Z := 1047,
	PCS_7_A := 1048,
	PCS_7_B := 1049,
	PCS_7_C := 1050,
	PCS_8_COORDTYPE := 1051,
	PCS_8_X := 1052,
	PCS_8_Y := 1053,
	PCS_8_Z := 1054,
	PCS_8_A := 1055,
	PCS_8_B := 1056,
	PCS_8_C := 1057,
	PCS_9_COORDTYPE := 1058,
	PCS_9_X := 1059,
	PCS_9_Y := 1060,
	PCS_9_Z := 1061,
	PCS_9_A := 1062,
	PCS_9_B := 1063,
	PCS_9_C := 1064,
	PCS_10_COORDTYPE := 1065,
	PCS_10_X := 1066,
	PCS_10_Y := 1067,
	PCS_10_Z := 1068,
	PCS_10_A := 1069,
	PCS_10_B := 1070,
	PCS_10_C := 1071,
	PCS_11_COORDTYPE := 1072,
	PCS_11_X := 1073,
	PCS_11_Y := 1074,
	PCS_11_Z := 1075,
	PCS_11_A := 1076,
	PCS_11_B := 1077,
	PCS_11_C := 1078,
	PCS_12_COORDTYPE := 1079,
	PCS_12_X := 1080,
	PCS_12_Y := 1081,
	PCS_12_Z := 1082,
	PCS_12_A := 1083,
	PCS_12_B := 1084,
	PCS_12_C := 1085,
	PCS_13_COORDTYPE := 1086,
	PCS_13_X := 1087,
	PCS_13_Y := 1088,
	PCS_13_Z := 1089,
	PCS_13_A := 1090,
	PCS_13_B := 1091,
	PCS_13_C := 1092,
	PCS_14_COORDTYPE := 1093,
	PCS_14_X := 1094,
	PCS_14_Y := 1095,
	PCS_14_Z := 1096,
	PCS_14_A := 1097,
	PCS_14_B := 1098,
	PCS_14_C := 1099,
	PCS_15_COORDTYPE := 1100,
	PCS_15_X := 1101,
	PCS_15_Y := 1102,
	PCS_15_Z := 1103,
	PCS_15_A := 1104,
	PCS_15_B := 1105,
	PCS_15_C := 1106,
	PCS_16_COORDTYPE := 1107,
	PCS_16_X := 1108,
	PCS_16_Y := 1109,
	PCS_16_Z := 1110,
	PCS_16_A := 1111,
	PCS_16_B := 1112,
	PCS_16_C := 1113,
	MCS_X := 1121,
	MCS_Y := 1122,
	MCS_Z := 1123,
	MCS_A := 1124,
	MCS_B := 1125,
	MCS_C := 1126,
	ACTIVETOOL := 1150,
	TOOL_1_TOOLTYPE := 1151,
	TOOL_1_X := 1152,
	TOOL_1_Y := 1153,
	TOOL_1_Z := 1154,
	TOOL_1_A := 1155,
	TOOL_1_B := 1156,
	TOOL_1_C := 1157,
	TOOL_1_SWITCHONTIME := 1158,
	TOOL_1_SWITCHOFFTIME := 1159,
	TOOL_2_TOOLTYPE := 1171,
	TOOL_2_X := 1172,
	TOOL_2_Y := 1173,
	TOOL_2_Z := 1174,
	TOOL_2_A := 1175,
	TOOL_2_B := 1176,
	TOOL_2_C := 1177,
	TOOL_2_SWITCHONTIME := 1178,
	TOOL_2_SWITCHOFFTIME := 1179,
	TOOL_3_TOOLTYPE := 1191,
	TOOL_3_X := 1192,
	TOOL_3_Y := 1193,
	TOOL_3_Z := 1194,
	TOOL_3_A := 1195,
	TOOL_3_B := 1196,
	TOOL_3_C := 1197,
	TOOL_3_SWITCHONTIME := 1198,
	TOOL_3_SWITCHOFFTIME := 1199,
	TOOL_4_TOOLTYPE := 1211,
	TOOL_4_X := 1212,
	TOOL_4_Y := 1213,
	TOOL_4_Z := 1214,
	TOOL_4_A := 1215,
	TOOL_4_B := 1216,
	TOOL_4_C := 1217,
	TOOL_4_SWITCHONTIME := 1218,
	TOOL_4_SWITCHOFFTIME := 1219,
	COULOMBFRICTIONA1 := 3051,
	COULOMBFRICTIONA2 := 3052,
	COULOMBFRICTIONA3 := 3053,
	COULOMBFRICTIONA4 := 3054,
	COULOMBFRICTIONA5 := 3055,
	COULOMBFRICTIONA6 := 3056,
	VISCOSEFRICTIONA1 := 3057,
	VISCOSEFRICTIONA2 := 3058,
	VISCOSEFRICTIONA3 := 3059,
	VISCOSEFRICTIONA4 := 3060,
	VISCOSEFRICTIONA5 := 3061,
	VISCOSEFRICTIONA6 := 3062,
	GRAVITATIONX := 3071,
	GRAVITATIONY := 3072,
	GRAVITATIONZ := 3073,
	MINIMALDYNAMICPARAMETER1 := 3074,
	MINIMALDYNAMICPARAMETER2 := 3075,
	MINIMALDYNAMICPARAMETER3 := 3076,
	MINIMALDYNAMICPARAMETER4 := 3077,
	MINIMALDYNAMICPARAMETER5 := 3078,
	MINIMALDYNAMICPARAMETER6 := 3079,
	MINIMALDYNAMICPARAMETER7 := 3080,
	MINIMALDYNAMICPARAMETER8 := 3081,
	MINIMALDYNAMICPARAMETER9 := 3082,
	MINIMALDYNAMICPARAMETER10 := 3083,
	MINIMALDYNAMICPARAMETER11 := 3084,
	MINIMALDYNAMICPARAMETER12 := 3085,
	MINIMALDYNAMICPARAMETER13 := 3086,
	MINIMALDYNAMICPARAMETER14 := 3087,
	MINIMALDYNAMICPARAMETER15 := 3088,
	MINIMALDYNAMICPARAMETER16 := 3089,
	MINIMALDYNAMICPARAMETER17 := 3090,
	MINIMALDYNAMICPARAMETER18 := 3091
);
END_TYPE

(* ---- L_MC4P_PATHDATA.dut ---- *)
TYPE L_MC4P_PATHDATA :
STRUCT
	RESERVED : ARRAY [1..SIZEOF(L_MC4P_AuxAxesData)] OF BYTE;
	VMAX_IN : LREAL;
	VMAX_OUT : LREAL;
	VMAX : LREAL;
	AMAX : LREAL;
	DMAX : LREAL;
	AMAX_ORIG : LREAL := L_UMTP_Math.L_UMTP_ValueInitial;
	DMAX_ORIG : LREAL := L_UMTP_Math.L_UMTP_ValueInitial;
	LRJERK : LREAL;
	ALRVMAXROT : ARRAY [1..3] OF LREAL;
	ALRAMAXROT : ARRAY [1..3] OF LREAL;
	ALRJERKROT : ARRAY [1..3] OF LREAL;
	VEL_IN_ROT : ARRAY [1..3] OF LREAL;
	VEL_OUT_ROT : ARRAY [1..3] OF LREAL;
	SCBLENDINGDATA : L_MC4P_BlendingData;
END_STRUCT
END_TYPE

(* ---- L_MC4P_PATHELEMENT.dut ---- *)
TYPE L_MC4P_PATHELEMENT :
STRUCT
	XDATAVALID : BOOL;
	ISETNO : DINT;
	ESEGMENTTYPE : L_MC4P_SegmentType;
	ALRTARGETPOS : ARRAY [1..12] OF LREAL;
	ALRTARGETPOSAUX : ARRAY [1..6] OF LREAL;
	ALRCENTERPOINT : ARRAY [1..12] OF LREAL;
	LRVELMAX : LREAL;
	LRACCMAX : LREAL;
	LRDECMAX : LREAL;
	LRJERK : LREAL;
	ALRVELROTMAX : ARRAY [1..3] OF LREAL;
	ALRACCROTMAX : ARRAY [1..3] OF LREAL;
	ALRJERKROT : ARRAY [1..3] OF LREAL;
	ALRVELOCITYPTP : ARRAY [1..6] OF LREAL;
	ALRACCELERATIONPTP : ARRAY [1..6] OF LREAL;
	ALRDECELERATIONPTP : ARRAY [1..6] OF LREAL;
	ALRJERKPTP : ARRAY [1..6] OF LREAL;
	XSMOOTHACTIVE : BOOL;
	LRSMOOTHTOLPERC : LREAL;
	LRSMOOTHRADIUS : LREAL;
	ESMOOTHTYPE : L_MC4P_SegmentType;
	BUFFERMODE : MC_BUFFER_MODE;
	AEAUXMODE : ARRAY [1..6] OF L_MC4P_AuxMode;
	ALRVELOCITYAUX : ARRAY [1..6] OF LREAL;
	ALRACCELERATIONAUX : ARRAY [1..6] OF LREAL;
	ALRDECELERATIONAUX : ARRAY [1..6] OF LREAL;
	ALRJERKAUX : ARRAY [1..6] OF LREAL;
	PATHCHOICE : MC_CIRC_PATHCHOICE;
	ALR_RN_CIRC : ARRAY [1..3] OF LREAL;
	LAMBDA_MAX : LREAL;
	RADIUS : LREAL;
	LENGTH : LREAL;
	R_S : ARRAY [1..3, 1..3] OF LREAL;
	LRSEMIMAJORAXIS : LREAL;
	LRSEMIMINORAXIS : LREAL;
	LRECCENTRICITY : LREAL;
	LRPHI0 : LREAL;
	LRPHI1 : LREAL;
	LRS0 : LREAL;
	LRS1 : LREAL;
	LRARCLENGTH0 : LREAL;
	LRWAITTIME : LREAL;
	SCTRAFOINFO : L_MC4P_TrafoInfo;
	ALRTOOLCHANGEOFFSET : ARRAY [1..3] OF LREAL;
	XWTRACKFBINSTANCE : __XWORD;
	ALRSTARTSUPERPOSPOS : ARRAY [1..3] OF LREAL;
	EORIENTATIONMODE : L_MC4P_Orientation_Mode;
	AEDIRECTION : ARRAY [1..6] OF MC_DIRECTION;
	UICNTINTERMEDIATEPOINTS : UINT;
	ASCSPLINEDATA : ARRAY [1..10] OF L_MC4P_SplineData;
	XDONTCALCPROFILEMOVEPATH : BOOL;
END_STRUCT
END_TYPE

(* ---- L_MC4P_PATHLISTDIAGNOSTICDATA.dut ---- *)
TYPE L_MC4P_PATHLISTDIAGNOSTICDATA :
STRUCT
	DITASKCOUNTERNOCHANGES : DINT;
	DITIMESTAMP : DINT;
	ADIELEMNTSEGMENTNO : ARRAY [1..30] OF DINT;
	ADWELEMNTMASK : ARRAY [1..30] OF DWORD;
	XEXECUTEPATHSTOP : BOOL;
	LROVERRIDE : LREAL := 1;
	DIFUNID : DINT;
	DIACTFUNID : DINT;
	DIBUSYFUNID : DINT;
END_STRUCT
END_TYPE

(* ---- L_MC4P_PATHREFMONITORDATA.dut ---- *)
TYPE L_MC4P_PATHREFMONITORDATA :
STRUCT
	EGCODETYPE : L_MC4P_GCodeType := L_MC4P_GCodeType.undefined;
	SSOURCELINE : STRING(255) := '';
	LIFILELINENO : LINT;
	LILINENO : LINT;
	ALRPOSDIST : ARRAY [1..12] OF LREAL;
	XRELATIVE : BOOL;
	ECOORDSYSTEM : L_MC4P_CoordSystem;
END_STRUCT
END_TYPE

(* ---- L_MC4P_PCSTRACKPARAM.dut ---- *)
TYPE L_MC4P_PCSTRACKPARAM :
STRUCT
	XWTRACKFBINSTANCE : __XWORD;
	XWTRACKINSTANCEACTIVE : __XWORD;
	XWINSTANCECALLBACK : __XWORD;
	XPCSVALID : BOOL;
	BSTOPTRIGGER : BOOL;
END_STRUCT
END_TYPE

(* ---- L_MC4P_POLYCHARACTERISTICS.dut ---- *)
TYPE L_MC4P_POLYCHARACTERISTICS :
STRUCT
	LRX : LREAL;
	LRY : LREAL;
	LRYS : LREAL;
	LRYSS : LREAL;
	LRA1 : LREAL;
	LRA2 : LREAL;
	LRA3 : LREAL;
	LRA4 : LREAL;
	LRA5 : LREAL;
END_STRUCT
END_TYPE

(* ---- L_MC4P_POLYNOMDATA.dut ---- *)
TYPE L_MC4P_POLYNOMDATA :
STRUCT
	RESERVED : ARRAY [1..SIZEOF(L_MC4P_PathData)] OF BYTE;
	ALRPATHKOEFF : ARRAY [1..3, 1..6] OF LREAL;
END_STRUCT
END_TYPE

(* ---- L_MC4P_PRECONTROLFRICTIONLOCATION.dut ---- *)
TYPE L_MC4P_PRECONTROLFRICTIONLOCATION :
(
	ACS := 1,
	JCS := 2
);
END_TYPE

(* ---- L_MC4P_PTPDATA.dut ---- *)
TYPE L_MC4P_PTPDATA :
STRUCT
	RESERVED : ARRAY [1..SIZEOF(L_MC4P_AuxAxesData)] OF BYTE;
	ALRPTPJERK : ARRAY [1..6] OF LREAL;
	ALRPTPACC : ARRAY [1..6] OF LREAL;
	ALRPTPVEL : ARRAY [1..6] OF LREAL;
	ALRPTPJERK_ORIGIN : ARRAY [1..6] OF LREAL;
	ALRPTPACC_ORIGIN : ARRAY [1..6] OF LREAL;
	ALRPTPVEL_ORIGIN : ARRAY [1..6] OF LREAL;
	LRPTP_MAXTIME : LREAL;
	PTPTYPE : ARRAY [1..6] OF L_MC4P_PTPTypes;
	VMAX_IN_PTP : ARRAY [1..6] OF LREAL;
	VMAX_OUT_PTP : ARRAY [1..6] OF LREAL;
END_STRUCT
END_TYPE

(* ---- L_MC4P_PTPPREPSTATES.dut ---- *)
TYPE L_MC4P_PTPPREPSTATES :
(
	IDENTTMAX := 100,
	IDENTPTPTYPE := 200,
	CALCPTPPROFILE := 300,
	QUITPREP := 900
);
END_TYPE

(* ---- L_MC4P_PTPTYPES.dut ---- *)
TYPE L_MC4P_PTPTYPES :
(
	NONE := 0,
	REDVMAX := 100,
	RAST2RAST := 200,
	RAST2VEL := 300,
	RAST2VEL_UNTERLAGERT := 350,
	VEL2RAST := 400,
	VEL2RAST_UNTERLAGERT := 450,
	VEL2VEL := 500
);
END_TYPE

(* ---- L_MC4P_SCPICKANDPLACEPROFILEPARBASE.dut ---- *)
TYPE L_MC4P_SCPICKANDPLACEPROFILEPARBASE :
STRUCT
	LRXPOS : LREAL;
	LRYPOS : LREAL;
	LRZPOS : LREAL;
	LRAPOS : LREAL := 180;
	LRBPOS : LREAL;
	LRCPOS : LREAL;
	LRAUX1POS : LREAL;
	LRPATHVEL : LREAL := 0;
	LRPATHACC : LREAL := 0;
	LRPATHDEC : LREAL := 0;
	LRBLENDINGRADIUS : LREAL := 0;
	XHALT : BOOL := FALSE;
	EORIENTATIONMODE : L_MC4P_Orientation_Mode := L_MC4P_Orientation_Mode.ShortestSpacialWay;
	EADIRECTION : MC_DIRECTION := MC_DIRECTION.mcShortestWay;
	EBDIRECTION : MC_DIRECTION := MC_DIRECTION.mcShortestWay;
	ECDIRECTION : MC_DIRECTION := MC_DIRECTION.mcShortestWay;
END_STRUCT
END_TYPE

(* ---- L_MC4P_SCPICKANDPLACEPROFILEPARSTATE.dut ---- *)
TYPE L_MC4P_SCPICKANDPLACEPROFILEPARSTATE :
STRUCT
	ECOORDSYSTEM : L_MC4P_CoordSystem := L_MC4P_CoordSystem.WCS;
END_STRUCT
END_TYPE

(* ---- L_MC4P_SEGMENTTYPE.dut ---- *)
TYPE L_MC4P_SEGMENTTYPE :
(
	UNDEF := 0,
	P1 := 1,
	P5 := 5,
	CIRC := 10,
	ELLIPSE := 20,
	CUBICSPLINE := 30,
	PTP := 100,
	WAITTIME := 200,
	GROUPSTOP := -1,
	STOPALL := -2
);
END_TYPE

(* ---- L_MC4P_SETVALUEFILTERMODE.dut ---- *)
TYPE L_MC4P_SETVALUEFILTERMODE :
(
	EQUALYSPACED := 1,
	SYMTRIANGLE := 2,
	GAUSSIANDISTRIBUTED_1SIGMA := 11,
	GAUSSIANDISTRIBUTED_2SIGMA := 12,
	GAUSSIANDISTRIBUTED_3SIGMA := 13,
	GAUSSIANDISTRIBUTED_4SIGMA := 14,
	HALFSINE := 21,
	ONEMINUSCOSINE := 22
);
END_TYPE

(* ---- L_MC4P_SKIPGCODE.dut ---- *)
TYPE L_MC4P_SKIPGCODE :
STRUCT
	XG00 : BOOL;
	XG01 : BOOL;
	XG02 : BOOL;
	XG03 : BOOL;
	XG04 : BOOL;
	XG16 : BOOL;
	XG17 : BOOL;
	XG18 : BOOL;
	XG19 : BOOL;
	XG22 : BOOL;
	XG50 : BOOL;
	XG51 : BOOL;
	XG53 : BOOL;
	XG54 : BOOL;
	XG55 : BOOL;
	XG56 : BOOL;
	XG57 : BOOL;
	XG58 : BOOL;
	XG59 : BOOL;
	XG75 : BOOL;
	XG90 : BOOL;
	XG91 : BOOL;
	XG98 : BOOL;
	XG99 : BOOL;
	XENDOFSUBROUTINE : BOOL;
	XENDOFPROGRAM : BOOL;
	XMOS : BOOL;
	XMVS_SVS : BOOL;
	XMVS_SNS : BOOL;
	XMNS_SNS : BOOL;
END_STRUCT
END_TYPE

(* ---- L_MC4P_SOURCEOFMOTIONCOMMAND.dut ---- *)
TYPE L_MC4P_SOURCEOFMOTIONCOMMAND :
(
	CONTPATHPREPARE := 16#1,
	MOVEPATH := 16#2,
	GROUPSTOP := 16#4,
	STOPALL := 16#8,
	QSP := 16#10,
	SINGLEWCS := 16#10000,
	COORDINATEDCP := 16#20000,
	MANMODEWCS := 16#40000,
	MANMODECARTESIAN := 16#80000,
	STOPWCS := 16#100000,
	WCSSETVALUEFILTER := 16#200000,
	TRACKING := 16#400000,
	SINGLEACS := 16#100000000,
	GROUPHOMINGACS := 16#200000000,
	MANMODEACS := 16#400000000,
	COORDINATEDPTP := 16#800000000,
	STOPACS := 16#1000000000,
	ANYWCSMOTION := 16#FFFF0000,
	ANYWCSMOTIONEXCEPTWCSFILTER := 16#FFDF0000,
	ANYACSMOTION := 16#FFFF00000000,
	ANYMOTION := 16#FFFFFFFF0000
);
END_TYPE

(* ---- L_MC4P_SPACEOFMOTION.dut ---- *)
TYPE L_MC4P_SPACEOFMOTION :
(
	JOINTSPACE := 1,
	TASKSPACE := 2
);
END_TYPE

(* ---- L_MC4P_SPLINEDATA.dut ---- *)
TYPE L_MC4P_SPLINEDATA :
STRUCT
	INPOINT : ARRAY [1..3] OF LREAL;
	INNUMBER : UINT;
	LSI : LREAL;
	LSICUMULATED : LREAL;
	LUICUMULATED : LREAL;
	PATHKOEFFSNORM : ARRAY [1..3, 1..4] OF LREAL;
END_STRUCT
END_TYPE

(* ---- L_MC4P_SUPERPOSHANDLER.dut ---- *)
TYPE L_MC4P_SUPERPOSHANDLER :
STRUCT
	DATAVALID : BOOL := FALSE;
	ALRSUPERPOSPOSCCS : ARRAY [1..6] OF LREAL;
	ALRSUPERPOSVELCCS : ARRAY [1..6] OF LREAL;
	ALRSUPERPOSACCCCS : ARRAY [1..6] OF LREAL;
	PTRAFO_BASE_WCS : POINTER TO L_MC4P_CoordTrafo;
	ETRACKINGTYPE : L_MC4P_TrackingFBTypes;
END_STRUCT
END_TYPE

(* ---- L_MC4P_SWITCHINGFUNCTIONDATA.dut ---- *)
TYPE L_MC4P_SWITCHINGFUNCTIONDATA :
STRUCT
	AISWITCHINGFUNID : ARRAY [1..L_MC4P_Constants.gciMaxNumParallelSwitchingFun] OF INT;
	ALRSWITCHINGFUNPARAM : ARRAY [1..L_MC4P_Constants.gciMaxNumParallelSwitchingFun] OF LREAL;
	AESWITCHINGFUNPARAMTYPE : ARRAY [1..L_MC4P_Constants.gciMaxNumParallelSwitchingFun] OF L_MC4P_SwitchingFunParamType;
END_STRUCT
END_TYPE

(* ---- L_MC4P_SWITCHINGFUNPARAMTYPE.dut ---- *)
TYPE L_MC4P_SWITCHINGFUNPARAMTYPE :
(
	UNDEFINED := 0,
	NORMEDPOS := 1,
	DISTFROMSTART := 2,
	DISTTOTARGET := 3,
	EVALUATED := 255
);
END_TYPE

(* ---- L_MC4P_TEACHCOORDINATESYSTEMSTEPS.dut ---- *)
TYPE L_MC4P_TEACHCOORDINATESYSTEMSTEPS :
(
	NONE := 0,
	TEACHORIGIN := 1,
	TEACHPOSXAXIS := 2,
	TEACHPOSQUADRANTXY := 3,
	DONE := 4
);
END_TYPE

(* ---- L_MC4P_TOOL_REF.dut ---- *)
TYPE L_MC4P_TOOL_REF :
STRUCT
	TOOLTYPE : L_MC4P_ToolType := L_MC4P_ToolType.Cartesian;
	X : LREAL;
	Y : LREAL;
	Z : LREAL;
	A : LREAL;
	B : LREAL;
	C : LREAL;
	SWITCHONTIME : LREAL;
	SWITCHOFFTIME : LREAL;
END_STRUCT
END_TYPE

(* ---- L_MC4P_TOOLREQUEST.dut ---- *)
TYPE L_MC4P_TOOLREQUEST :
(
	HOLD := 0,
	ON := 1,
	OFF := 2
);
END_TYPE

(* ---- L_MC4P_TOOLSYSTEM.dut ---- *)
TYPE L_MC4P_TOOLSYSTEM :
(
	NOTOOL := 0,
	TOOL_1 := 1,
	TOOL_2 := 2,
	TOOL_3 := 3,
	TOOL_4 := 4
);
END_TYPE

(* ---- L_MC4P_TOOLTYPE.dut ---- *)
TYPE L_MC4P_TOOLTYPE :
(
	CARTESIAN := 0
);
END_TYPE

(* ---- L_MC4P_TRACKINGDATA.dut ---- *)
TYPE L_MC4P_TRACKINGDATA :
STRUCT
	XWTRACKFBINSTANCE : __XWORD;
	ALRSTARTSUPERPOSPOS : ARRAY [1..3] OF LREAL;
END_STRUCT
END_TYPE

(* ---- L_MC4P_TRACKINGFBTYPES.dut ---- *)
TYPE L_MC4P_TRACKINGFBTYPES :
(
	CONVEYORTRACKING := 0,
	ROTARYTRACKING := 1
);
END_TYPE

(* ---- L_MC4P_TRACKINGHANDSHAKE.dut ---- *)
TYPE L_MC4P_TRACKINGHANDSHAKE :
STRUCT
	XWACTIVETRACKFBINST : __XWORD;
	XRESTARTSYNC : BOOL;
	XWTRACKFBINSTTOCALCINITPCS : __XWORD;
	XLOOKFWDNOTABORTING : BOOL;
	XWTRACKINSTSYNCOUTREQUESTED : __XWORD;
	XTRACKINGABORTACTIVE : BOOL;
	ALRSUPERPOSPOSMCS : ARRAY [1..3] OF LREAL;
	ALRSUPERPOSVELMCS : ARRAY [1..3] OF LREAL;
	ALRSUPERPOSACCMCS : ARRAY [1..3] OF LREAL;
END_STRUCT
END_TYPE

(* ---- L_MC4P_TRACKINPUTPARAM.dut ---- *)
TYPE L_MC4P_TRACKINPUTPARAM :
STRUCT
	LRCLUTCHDISTANCE : LREAL;
	LRCLUTCHTIME : LREAL;
	LRCLUTCHTIMEABORT : LREAL;
	ALRINITMASTERPOS : ARRAY [1..6] OF LREAL;
	SCCOORDREF_INITOBJ_BASE : MC_Coord_Ref;
	SCTRAFO_BASE_MCS : L_MC4P_CoordTrafo;
	PTRACKINGCOORDPARAM : POINTER TO L_MC4P_PCSTrackParam;
	PCOORDTRAFO : POINTER TO L_MC4P_CoordTrafo;
END_STRUCT
END_TYPE

(* ---- L_MC4P_TRACKKINEMATICSSTATES.dut ---- *)
TYPE L_MC4P_TRACKKINEMATICSSTATES :
(
	INITIAL := 0,
	WAITFORMOTION := 250,
	SYNCIN := 500,
	SYNCHRON := 1000,
	SYNCOUT := 1500,
	AGSTOP := 2000,
	ABORTING := 8888,
	ERRORSTATE := 9999
);
END_TYPE

(* ---- L_MC4P_VISULISTTABLEDATA.dut ---- *)
TYPE L_MC4P_VISULISTTABLEDATA :
STRUCT
	DISEGMENTNO : DINT;
	DISEGMENTNOCOPIEDFROM : DINT;
	DWMASK : DWORD;
	XWAITINGFORPROFILEPREP : BOOL;
	SFBINSTANCE : STRING;
	ACT_T : LREAL;
	PLISTELEMENT : POINTER TO L_MC4P_ListElement;
	PATHLENGTH : LREAL;
	VINXYZ : LREAL;
	VMAXXYZ : LREAL;
	VOUTXYZ : LREAL;
	DELTAC : LREAL;
	VINC : LREAL;
	VMAXC : LREAL;
	VOUTC : LREAL;
END_STRUCT
END_TYPE

(* ---- L_MC4P_WAITTIMEDATA.dut ---- *)
TYPE L_MC4P_WAITTIMEDATA :
STRUCT
	LRWAITTIME : LREAL;
END_STRUCT
END_TYPE

(* ---- L_MC4P_WORKPIECEDATABASE.dut ---- *)
TYPE L_MC4P_WORKPIECEDATABASE :
STRUCT
	DWMASK : DWORD;
	WOJECTADRNO : WORD;
	WWORKPIECEID : WORD;
	XVALIDPOS : BOOL;
	ALROBJECTPOSITION : ARRAY [1..6] OF LREAL;
	LRAUX1TARGETPOS : LREAL;
	ALRDATA : ARRAY [1..12] OF LREAL;
	AIDATA : ARRAY [1..12] OF INT;
END_STRUCT
END_TYPE

(* ---- L_MC4P_WORKPIECEDATAINTERNALBASE.dut ---- *)
TYPE L_MC4P_WORKPIECEDATAINTERNALBASE :
STRUCT
	XINIT : BOOL;
	XRESERVE : BOOL;
	XWORKPIECEONBELTRECEIVE : BOOL;
	XVALIDPOS : BOOL;
	XPOSOUTOFLOWERLIMIT : BOOL;
	XPOSOUTOFUPPERLIMIT : BOOL;
	XPOSINWINDOW : BOOL;
	IMODULOPOS : UINT;
	LRAXISPOS : LREAL;
	LRINITIALXPOS : LREAL;
	LRDIST : LREAL;
	LRUPPERSYNCLIMIT : LREAL;
	LRLOWERSYNCLIMIT : LREAL;
	LRRESTDISTINWINDOW : LREAL;
	LRRESTDISTTOWINDOW : LREAL;
	LRRESTTIMEPOSINWINDOW : LREAL;
	LRRESTTIMEPOSTOWINDOW : LREAL;
END_STRUCT
END_TYPE

(* ---- MC_CIRC_PATHCHOICE.dut ---- *)
TYPE MC_CIRC_PATHCHOICE :
(
	CLOCKWISE := 0,
	COUNTERCLOCKWISE := 1
);
END_TYPE

(* ---- MC_COORD_REF.dut ---- *)
TYPE MC_COORD_REF :
STRUCT
	COORDTYPE : L_MC4P_CoordType := L_MC4P_CoordType.Cartesian;
	X : LREAL;
	Y : LREAL;
	Z : LREAL;
	A : LREAL;
	B : LREAL;
	C : LREAL;
END_STRUCT
END_TYPE

(* ---- MC_TRANSITION_MODE.dut ---- *)
TYPE MC_TRANSITION_MODE :
(
	TMNONE := 0,
	TMCORNERDISTANCE := 3
);
END_TYPE

(* ---- VISULISTTABLEDATA.dut ---- *)
TYPE VISULISTTABLEDATA :
STRUCT
	ISEGMENTNO : INT;
	SFBINSTANCE : STRING;
	ACT_T : LREAL;
	DWMASK : DWORD;
	TEST_01 : DINT;
	TEST_02 : DINT;
	TEST_03 : DINT;
	TEST_04 : DINT;
	TEST_05 : DINT;
	TEST_06 : DINT;
END_STRUCT
END_TYPE

(* ---- GVL_MATH.gvl ---- *)
VAR_GLOBAL
	EPS_ORI_THETA_PROFILE : LREAL := 1E-05;
END_VAR

(* ---- GVL_MOVEPATH.gvl ---- *)
VAR_GLOBAL
	GCINUMOFDECODEASCIIDATA : INT := 30;
	GCINUMOFDECODEASCIIDATA_RESERVE : INT := 5;
	GCINUMOFPATHFILES : INT := 5;
END_VAR

(* ---- GVL_MOVESPLINE.gvl ---- *)
VAR_GLOBAL
	LENGTHVEC_SPLINE : UINT := 101;
	MAXINTERMEDIATEPOINTS : UINT := 9;
END_VAR

(* ---- GVL_TEST.gvl ---- *)
VAR_GLOBAL
	ADWTRACKINGCASECOUNTER : ARRAY [1..20] OF DWORD := [20(0)];
	DWLASTTRACKINGCASE : DWORD;
	GDWUNDOBLENDINGCOUNTER : DWORD;
	GPAGDIRCREATE : POINTER TO AXES_GROUP_KIN;
	GXDIRCREATEMOVEPATHDATADONE : BOOL;
	GXDIRCREATEMOVEPATHDATABUSY : BOOL;
	GXDIRCREATEDIAGNOSISDATADONE : BOOL;
	GXDIRCREATEDIAGNOSISDATABUSY : BOOL;
	GULITIMESTART : ULINT;
	GULITIMEEND : ULINT;
	GAULIDURATION : ARRAY [1..20] OF ULINT;
	GCSAVEIPOMONITORINGERROR : BOOL := TRUE;
	GIELLIPSEINTERPOLATIONCHOICE : INT := 3;
END_VAR

(* ---- L_MC4P_CONSTANTS.gvl ---- *)
VAR_GLOBAL
	LENGTHVEC_IDXMAX : UINT := 1001;
	BENDING_IDXMAX : INT := 51;
	NULLVEKTOR3D : ARRAY [1..3] OF LREAL := [0, 0, 0];
	SIZEVISUARRAY : WORD := 30;
	PUDILISTSEMACONST : POINTER TO Systypes.RTS_IEC_RESULT := 0;
	MAXCOUNTLISTELEMENTS : INT := 100;
	GCWLA_HORIZONPTP : WORD := 1;
	UIMAXNBROFDYNAMICPAR : UINT := 24;
	GCUSIMAXFOURIERCOEFFSIDENT : USINT := 5;
	CINUMOFMOVECONTPATH : INT := 30;
	GCIMAXNUMPARALLELMFUN : INT := 10;
	GCIMAXNUMPARALLELSWITCHINGFUN : INT := 3;
END_VAR

(* ---- L_MC4P_INTERNAL.gvl ---- *)
VAR_GLOBAL
	CDIENUMSTARTVALUE : DINT := 70000;
END_VAR

(* ---- LUT_ELLIPTICALINTEGRAL.gvl ---- *)
VAR_GLOBAL
	GCUIELLIPTICINTEGRAL_DIMEPS : UINT := 101;
	GCUIELLIPTICINTEGRAL_DIMT : UINT := 1001;
	GALRELLIPTICINTEGRAL : ARRAY [1..LUT_EllipticalIntegral.gcuiEllipticIntegral_DimEps, 1..LUT_EllipticalIntegral.gcuiEllipticIntegral_Dimt] OF LREAL;
	GALRELLIPTICINTEGRALEPSILON : ARRAY [1..LUT_EllipticalIntegral.gcuiEllipticIntegral_DimEps] OF LREAL := [0, 0.045462034321782, 0.0888779400445358, 0.13033980812517099, 0.169935584744777, 0.207749257854261, 0.243861035324057, 0.278347515075767, 0.31128184755663, 0.342733890901418, 0.372770359110916, 0.401454963561255, 0.428848548144286, 0.455009218325632, 0.479992464394169, 0.503851279164371, 0.526636270381173, 0.548395768065783, 0.569175927030135, 0.589020824777439, 0.607972554996467, 0.626071316847918, 0.643355500232221, 0.659861767219665, 0.675625129815564, 0.690679024225416, 0.705055381777574, 0.718784696653878, 0.731896090571903, 0.744417374556022, 0.756375107928325, 0.767794654644496, 0.778700237094164, 0.789114987479843, 0.79906099688343, 0.808559362124356, 0.817630230508763, 0.826292842564648, 0.834565572853598, 0.842465968945701, 0.850010788640292, 0.857216035511494, 0.864096992853947, 0.870668256100719, 0.876943763782181, 0.882936827091498, 0.888660158119453, 0.894125896818497, 0.899345636753214, 0.904330449691828, 0.909090909090909, 0.913637112523087, 0.917978703095363, 0.922124889903426, 0.926084467565387, 0.929865834876335, 0.933477012623315, 0.936925660598486, 0.940219093846572, 0.943364298181051, 0.946367945002001, 0.949236405447035, 0.951975763905338, 0.954591830923472, 0.957090155530326, 0.959476037007346, 0.961754536129027, 0.963930485897487, 0.966008501793923, 0.967992991568653, 0.969888164590556, 0.971698040775701, 0.973426459114131, 0.975077085812876, 0.976653422072466, 0.978158811513451, 0.979596447268666, 0.980969378756297, 0.982280518148099, 0.983532646546511, 0.984728419883742, 0.985870374555359, 0.986960932800325, 0.988002407838893, 0.988997008779252, 0.989946845303345, 0.990853932141785, 0.991720193347374, 0.992547466376269, 0.993337505985479, 0.994091987954938, 0.99481251264205794, 0.995500608376304, 0.996157734700981, 0.996785285469127, 0.997384591800059, 0.997956924902854, 0.998503498772759, 0.999025472766231, 0.999523954060092, 1];
	GLRELLIPTICALTARGETTOLERANCE : LREAL := 0.1;
END_VAR

(* ---- L_MC4P_DYNAMICPAR.itf ---- *)
INTERFACE L_MC4P_DYNAMICPAR
END_INTERFACE

METHOD GETDYNAMICPAR : L_IE1P_Error
VAR_IN_OUT
	AXESGROUP : AXES_GROUP_KIN;
	ALRDYNAMICPAR : ARRAY [1..L_MC4P_Constants.uimaxNbrOfDynamicPar] OF LREAL;
END_VAR
END_METHOD

METHOD GETFRICTION : L_IE1P_Error
VAR_IN_OUT
	AXESGROUP : AXES_GROUP_KIN;
	ALRVISCFRIC : ARRAY [1..6] OF LREAL;
	ALRCOULOMBFRIC : ARRAY [1..6] OF LREAL;
END_VAR
END_METHOD

METHOD GETGRAVITATION : L_IE1P_Error
VAR_IN_OUT
	AXESGROUP : AXES_GROUP_KIN;
	ALRGRAVITATION : ARRAY [1..3] OF LREAL;
END_VAR
END_METHOD

METHOD PARAMETERVALID : L_IE1P_Error
VAR_IN_OUT
	AXESGROUP : AXES_GROUP_KIN;
END_VAR
END_METHOD

(* ---- L_MC4P_IAXESGROUPMOTIONCOMMAND.itf ---- *)
INTERFACE L_MC4P_IAXESGROUPMOTIONCOMMAND
END_INTERFACE

METHOD ISACTIVEMOTIONCOMMAND : BOOL
VAR_INPUT
	ESRCOFCMD : L_MC4P_SourceOfMotionCommand;
END_VAR
END_METHOD

METHOD RELEASEMOTIONCOMMAND : BOOL
VAR_INPUT
	ESRCOFCMD : L_MC4P_SourceOfMotionCommand;
END_VAR
END_METHOD

METHOD REQUESTMOTIONCOMMAND : L_IE1P_Error
VAR_INPUT
	ESRCOFCMD : L_MC4P_SourceOfMotionCommand;
END_VAR
END_METHOD

METHOD RESETSOURCEOFMOTION
END_METHOD

(* ---- L_MC4P_ICLUTCH.itf ---- *)
INTERFACE L_MC4P_ICLUTCH
END_INTERFACE

METHOD CYCLECLUTCH : L_MC4P_TrackKinematicsStates
VAR_INPUT
	SCMASTER : L_MC4P_AxisProfile;
END_VAR
VAR_OUTPUT
	EERRORID : L_IE1P.L_IE1P_Error;
END_VAR
END_METHOD

METHOD GETACTUALMASTER
VAR_OUTPUT
	SCACTUALMASTER : L_MC4P_AxisProfile;
	EERRORID : L_IE1P.L_IE1P_Error;
END_VAR
END_METHOD

METHOD GETACTUALSLAVE
VAR_OUTPUT
	PACTUALSLAVE : POINTER TO L_MC4P_AxisProfile;
	DWSLAVECOUNT : DWORD;
	EERRORID : L_IE1P.L_IE1P_Error;
END_VAR
END_METHOD

METHOD STARTCLUTCH
VAR_INPUT
	LRMASTERSTART : LREAL;
	LRCYCLELENGTH : LREAL;
	LRSLAVEFINAL : LREAL;
	LRGEARRATIO : LREAL;
	LRCLUTCHDISTANCE : LREAL;
	ECLUTCHDIR : MC_DIRECTION;
	PSLAVESTART : POINTER TO L_MC4P_AxisProfile;
	DWSLAVECOUNT : DWORD;
END_VAR
VAR_OUTPUT
	EERRORID : L_IE1P.L_IE1P_Error;
END_VAR
END_METHOD

METHOD STOPCLUTCH
VAR_INPUT
	LRDECLUTCHDISTANCE : LREAL;
END_VAR
END_METHOD

(* ---- L_MC4P_IDIGSWITCHHANDLING.itf ---- *)
INTERFACE L_MC4P_IDIGSWITCHHANDLING
END_INTERFACE

METHOD CYCLICIPOCALL : BOOL
VAR_INPUT
	PLISTELEMENT : POINTER TO L_MC4P_ListElement;
	RSCCYCLICDATA : REFERENCE TO L_MC4P_CyclicData;
END_VAR
END_METHOD

METHOD FINALIZESEGMENT : BOOL
VAR_INPUT
	PLISTELEMENTACT : POINTER TO L_MC4P_ListElement;
	PLISTELEMENTNEXT : POINTER TO L_MC4P_ListElement;
END_VAR
END_METHOD

(* ---- L_MC4P_IDYNLIMITPROVIDER.itf ---- *)
INTERFACE L_MC4P_IDYNLIMITPROVIDER
END_INTERFACE

METHOD GETMAXACCELERATION : LREAL
VAR_INPUT
	IDX : UINT;
	EMAXVALUESOURCE : L_MC4P_MaxValueSource;
END_VAR
END_METHOD

METHOD GETMAXDECELERATION : LREAL
VAR_INPUT
	IDX : UINT;
	EMAXVALUESOURCE : L_MC4P_MaxValueSource;
END_VAR
END_METHOD

METHOD GETMAXJERK : LREAL
VAR_INPUT
	IDX : UINT;
	EMAXVALUESOURCE : L_MC4P_MaxValueSource;
END_VAR
END_METHOD

METHOD GETMAXVELOCITY : LREAL
VAR_INPUT
	IDX : UINT;
	EMAXVALUESOURCE : L_MC4P_MaxValueSource;
END_VAR
END_METHOD

(* ---- L_MC4P_IGEOOBJECT.itf ---- *)
INTERFACE L_MC4P_IGEOOBJECT
END_INTERFACE

METHOD BENDING : BOOL
VAR_INPUT
	LRPATHPOS : LREAL;
END_VAR
VAR_OUTPUT
	LRBENDING : LREAL;
	SCERROR : L_MC4P_ErrorStruct;
END_VAR
END_METHOD

METHOD CUT : BOOL
VAR_INPUT
	LRS0 : LREAL;
	LRS1 : LREAL;
END_VAR
VAR_OUTPUT
	SCERROR : L_MC4P_ErrorStruct;
END_VAR
END_METHOD

METHOD EXPANDLISTELEMENT : BOOL
VAR_OUTPUT
	SCERROR : L_MC4P_ErrorStruct;
END_VAR
END_METHOD

METHOD FINALIZE : BOOL
END_METHOD

METHOD GETFINALSETPOINTDATA : BOOL
VAR_OUTPUT
	SCERROR : L_MC4P_ErrorStruct;
END_VAR
VAR_IN_OUT
	SCSP : L_MC4P_CyclicData;
END_VAR
END_METHOD

METHOD GETINSTANCE : REFERENCE TO L_MC4P_GeoObjectInst
END_METHOD

METHOD GETLISTELEMENTDATA : REFERENCE TO L_MC4P_ListElementData
END_METHOD

METHOD GETSETPOINDATA : BOOL
VAR_OUTPUT
	SCERROR : L_MC4P_ErrorStruct;
END_VAR
VAR_IN_OUT
	SCSP : L_MC4P_CyclicData;
END_VAR
END_METHOD

METHOD MAPTOPATHCOORDINATE : BOOL
VAR_OUTPUT
	SCERROR : L_MC4P_ErrorStruct;
END_VAR
END_METHOD

METHOD UPDATEBOUNDS : BOOL
VAR_OUTPUT
	SCERROR : L_MC4P_ErrorStruct;
END_VAR
END_METHOD

METHOD WRITETOFILE : BOOL
VAR_INPUT
	SPATH : STRING;
END_VAR
END_METHOD

(* ---- L_MC4P_IJACOBI.itf ---- *)
INTERFACE L_MC4P_IJACOBI
END_INTERFACE

METHOD CALCDINVERSEJACOBIAN : BOOL
VAR_INPUT
	ICOORDPROVIDER : L_MC4P_IKinCoordProvider;
	PDINVJACOBIAN : POINTER TO ARRAY [1..6, 1..6] OF LREAL;
END_VAR
VAR_OUTPUT
	SCERROR : L_MC4P_ErrorStruct;
END_VAR
END_METHOD

METHOD CALCDJACOBIAN : BOOL
VAR_INPUT
	ICOORDPROVIDER : L_MC4P_IKinCoordProvider;
	PDJACOBIAN : POINTER TO ARRAY [1..6, 1..6] OF LREAL;
END_VAR
VAR_OUTPUT
	SCERROR : L_MC4P_ErrorStruct;
END_VAR
END_METHOD

METHOD CALCINVERSEJACOBIAN : BOOL
VAR_INPUT
	ICOORDPROVIDER : L_MC4P_IKinCoordProvider;
	PINVJACOBIAN : POINTER TO ARRAY [1..6, 1..6] OF LREAL;
END_VAR
VAR_OUTPUT
	SCERROR : L_MC4P_ErrorStruct;
END_VAR
END_METHOD

METHOD CALCJACOBIAN : BOOL
VAR_INPUT
	ICOORDPROVIDER : L_MC4P_IKinCoordProvider;
	PJACOBIAN : POINTER TO ARRAY [1..6, 1..6] OF LREAL;
END_VAR
VAR_OUTPUT
	SCERROR : L_MC4P_ErrorStruct;
END_VAR
END_METHOD

(* ---- L_MC4P_IKINCOORDPROVIDER.itf ---- *)
INTERFACE L_MC4P_IKINCOORDPROVIDER
END_INTERFACE

METHOD EQUALS : BOOL
VAR_INPUT
	ITFPROVIDER : L_MC4P_IKinCoordProvider;
	UDISYSTEM : UDINT;
	XPOS : BOOL;
	XVEL : BOOL;
	XACC : BOOL;
END_VAR
END_METHOD

(* ---- L_MC4P_IKINEMATICPARAMETER.itf ---- *)
INTERFACE L_MC4P_IKINEMATICPARAMETER
END_INTERFACE

METHOD CALCULATEPARAMETER
END_METHOD

METHOD CHECKPARAMETER : BOOL
END_METHOD

(* ---- L_MC4P_IKINPARAMEXTERN.itf ---- *)
INTERFACE L_MC4P_IKINPARAMEXTERN
END_INTERFACE

METHOD CALCULATEPARAMETER
END_METHOD

METHOD CHECKPARAMETER : BOOL
END_METHOD

(* ---- L_MC4P_IPATHELMDELETE.itf ---- *)
INTERFACE L_MC4P_IPATHELMDELETE
END_INTERFACE

METHOD CANCELFINISH
VAR_INPUT
	EERRORID : L_IE1P_Error;
END_VAR
END_METHOD

METHOD PREPAREFINISH
VAR_INPUT
	PLISTELMORIG : POINTER TO L_MC4P_ListElement;
	PLISTELMMODIFIED : POINTER TO L_MC4P_ListElement;
END_VAR
END_METHOD

(* ---- L_MC4P_IRESETABLE.itf ---- *)
INTERFACE L_MC4P_IRESETABLE
END_INTERFACE

METHOD RESET : BOOL
VAR_INPUT
	PBYSTATE : POINTER TO BYTE;
	UDISIZE : UDINT;
END_VAR
VAR_OUTPUT
	SCERROR : L_MC4P_ErrorStruct;
END_VAR
END_METHOD

METHOD STORESTATE : BOOL
VAR_INPUT
	PBYSTATE : POINTER TO BYTE;
	UDISIZE : UDINT;
END_VAR
VAR_OUTPUT
	SCERROR : L_MC4P_ErrorStruct;
END_VAR
END_METHOD

(* ---- L_MC4P_ITFEXTDYNAMICS.itf ---- *)
INTERFACE L_MC4P_ITFEXTDYNAMICS
END_INTERFACE

METHOD CALCEXTACSTORQUE
VAR_INPUT
	ALRACSPOS : ARRAY [1..6] OF LREAL;
	ALRACSVEL : ARRAY [1..6] OF LREAL;
	ALRACSACC : ARRAY [1..6] OF LREAL;
END_VAR
VAR_OUTPUT
	ALREXTTORQUE : ARRAY [1..6] OF LREAL;
END_VAR
END_METHOD

(* ---- L_MC4P_ITFTORQUEPRECONTROL.itf ---- *)
INTERFACE L_MC4P_ITFTORQUEPRECONTROL
END_INTERFACE

METHOD CARTESIANVALUESNEEDED : BOOL
END_METHOD

METHOD COPYTOPERSISTANTPARAMETER
END_METHOD

METHOD ENABLEINIT
VAR_IN_OUT
	AXESGROUP : AXES_GROUP_KIN;
END_VAR
END_METHOD

METHOD GETCYCLICDATA
VAR_IN_OUT
	ALRSETTORQUEOUT : ARRAY [1..6] OF LREAL;
END_VAR
END_METHOD

METHOD GETPERSISTANTPARAMETER
VAR_IN_OUT
	ALRDYNAMICPAR : ARRAY [1..L_MC4P_Constants.uimaxNbrOfDynamicPar] OF LREAL;
	ALRGRAVITATION : ARRAY [1..3] OF LREAL;
	ALRCOULOMBFRIC : ARRAY [1..6] OF LREAL;
	ALRVISCFRIC : ARRAY [1..6] OF LREAL;
END_VAR
END_METHOD

METHOD PARAMETERVALID : BOOL
VAR_IN_OUT
	AXESGROUP : AXES_GROUP_KIN;
	ALRDYNAMICPAR : ARRAY [1..L_MC4P_Constants.uimaxNbrOfDynamicPar] OF LREAL;
	ALRGRAVITATION : ARRAY [1..3] OF LREAL;
	ALRCOULOMBFRIC : ARRAY [1..6] OF LREAL;
	ALRVISCFRIC : ARRAY [1..6] OF LREAL;
END_VAR
END_METHOD

METHOD SETCYCLICPARAMETER
VAR_INPUT
	LRLOADMASS : LREAL;
	LRTOOLMASS : LREAL;
	ALRLOADINERTIA : ARRAY [1..3, 1..3] OF LREAL;
	ALRTOOLINERTIA : ARRAY [1..3, 1..3] OF LREAL;
	LRTORQUEOVERRIDE : LREAL;
	LRTORQUELIMITFACTOR : LREAL;
END_VAR
VAR_IN_OUT
	ALRTORQUEDELTACYCLE : ARRAY [1..6] OF LREAL;
END_VAR
END_METHOD

METHOD SETGRAVITATION
VAR_IN_OUT
	ALRGRAVITATION : ARRAY [1..3] OF LREAL;
END_VAR
END_METHOD

METHOD SETINITIALPARAMETER
VAR_INPUT
	XUSEFILTEREDVALUES : BOOL;
	EBEHAVEONERRORSTOP : L_MC4P_ErrorStopBehaviour;
	EFRICTIONLOCATION : L_MC4P_PreControlFrictionLocation;
END_VAR
VAR_IN_OUT
	ALRCOULOMBFRIC : ARRAY [1..6] OF LREAL;
	ALRVISCFRIC : ARRAY [1..6] OF LREAL;
	ALRDYNAMICPAR : ARRAY [1..L_MC4P_Constants.uimaxNbrOfDynamicPar] OF LREAL;
	ALRTORQUELIMITS : ARRAY [1..6] OF LREAL;
END_VAR
END_METHOD

METHOD CALCSETTORQUE
VAR_INPUT
	XENABLE : BOOL;
END_VAR
VAR_OUTPUT
	XBUSY : BOOL;
	SCERROR : L_MC4P_ErrorStruct;
END_VAR
VAR_IN_OUT
	AXESGROUP : AXES_GROUP_KIN;
	ALRSETTORQUE : ARRAY [1..6] OF LREAL;
END_VAR
END_METHOD

METHOD CALCULATEREGRESSIONMATRIX
VAR_INPUT
	EIDENTMODE : L_MC4P_IdentMode;
	USICYCLE : USINT;
END_VAR
VAR_IN_OUT
	ALRFLANGE_POS : ARRAY [1..6] OF LREAL;
	ALRFLANGE_VEL : ARRAY [1..6] OF LREAL;
	ALRFLANGE_ACC : ARRAY [1..6] OF LREAL;
	ALRJOINT_POS : ARRAY [1..6] OF LREAL;
	ALRJOINT_VEL : ARRAY [1..6] OF LREAL;
	ALRJOINT_ACC : ARRAY [1..6] OF LREAL;
END_VAR
END_METHOD

METHOD GETIDENTDATA
VAR_OUTPUT
	USINUMBEROFIDENTCYCLES : USINT;
	PLRPARAMETERVECTOR : POINTER TO LREAL;
	PLRPARAMETERVECTORMIN : POINTER TO LREAL;
	PLRPARAMETERVECTORMAX : POINTER TO LREAL;
	PASCIDENTTRAJ : POINTER TO ARRAY [1..6] OF L_MC4P_IdentTrajectoryFourierParam;
END_VAR
END_METHOD

METHOD GETIDENTIFIEDPARAMS
VAR_INPUT
	USICYCLE : USINT;
END_VAR
VAR_IN_OUT
	ALRDYNAMICPAR : ARRAY [1..L_MC4P_Constants.uimaxNbrOfDynamicPar] OF LREAL;
	ALRVISCFRIC : ARRAY [1..6] OF LREAL;
	ALRCOULOMBFRIC : ARRAY [1..6] OF LREAL;
END_VAR
END_METHOD

METHOD GETNUMBEROFDYNPARAMS : USINT
VAR_INPUT
	EIDENTMODE : L_MC4P_IdentMode;
	USICYCLE : USINT;
END_VAR
END_METHOD

METHOD GETREGRESSIONMATRIX
VAR_OUTPUT
	PLRREGRESSIONMATRIX : POINTER TO LREAL;
END_VAR
END_METHOD

METHOD GETSPACEOFMOTION : L_MC4P_SpaceOfMotion
END_METHOD

METHOD IDENTSUPPORTED : BOOL
END_METHOD

METHOD INITIDENTTRAJANDPARAMS
VAR_INPUT
	USICYCLE : USINT;
	XLIMITSAVAILABLE : BOOL;
END_VAR
VAR_IN_OUT
	ALRCOULOMBFRICMIN : ARRAY [1..6] OF LREAL;
	ALRVISCFRICMIN : ARRAY [1..6] OF LREAL;
	ALRDYNAMICPARMIN : ARRAY [1..L_MC4P_Constants.uimaxNbrOfDynamicPar] OF LREAL;
	ALRCOULOMBFRICMAX : ARRAY [1..6] OF LREAL;
	ALRVISCFRICMAX : ARRAY [1..6] OF LREAL;
	ALRDYNAMICPARMAX : ARRAY [1..L_MC4P_Constants.uimaxNbrOfDynamicPar] OF LREAL;
	ALRMINPOS : ARRAY [1..6] OF LREAL;
	ALRMAXPOS : ARRAY [1..6] OF LREAL;
END_VAR
END_METHOD

METHOD JOINTVALUESNEEDED : BOOL
END_METHOD

METHOD SETPARAMETERVECTOR
VAR_IN_OUT
	ALRDYNAMICPAR : ARRAY [1..L_MC4P_Constants.uimaxNbrOfDynamicPar] OF LREAL;
	ALRVISCFRIC : ARRAY [1..6] OF LREAL;
	ALRCOULOMBFRIC : ARRAY [1..6] OF LREAL;
END_VAR
END_METHOD

(* ---- L_MC4P_ITOOLINFO.itf ---- *)
INTERFACE L_MC4P_ITOOLINFO
END_INTERFACE

(* ---- L_MC4P_ITRAFOEXTENSION.itf ---- *)
INTERFACE L_MC4P_ITRAFOEXTENSION
END_INTERFACE

METHOD BACKWARDTRANSFORMATIONEXTENSION : L_IE1P_Error
VAR_INPUT
	PAXES_POS : POINTER TO ARRAY [1..6] OF LREAL;
	PJOINT_POS : POINTER TO ARRAY [1..6] OF LREAL;
END_VAR
END_METHOD

METHOD CHECKINPUTS : L_IE1P_Error
VAR_IN_OUT
	AXESGROUP : AXES_GROUP_KIN;
END_VAR
END_METHOD

METHOD FORWARDTRANSFORMATIONEXTENSION : L_IE1P_Error
VAR_INPUT
	PAXES_POS : POINTER TO ARRAY [1..6] OF LREAL;
	PJOINT_POS : POINTER TO ARRAY [1..6] OF LREAL;
END_VAR
END_METHOD

(* ---- L_MC4P_ITRAFOEXTERN.itf ---- *)
INTERFACE L_MC4P_ITRAFOEXTERN
END_INTERFACE

METHOD CALCBACKWARDTRAFO : WORD
VAR_IN_OUT
	AXESGROUP : AXES_GROUP_KIN;
	ALRPOSFLANGE : ARRAY [1..6] OF LREAL;
	ALRPOSAXES : ARRAY [1..6] OF LREAL;
	AICONFIGURATION : ARRAY [1..6] OF INT;
END_VAR
END_METHOD

METHOD CALCFORWARDTRAFO : WORD
VAR_IN_OUT
	AXESGROUP : AXES_GROUP_KIN;
	ALRPOSFLANGE : ARRAY [1..6] OF LREAL;
	ALRPOSAXES : ARRAY [1..6] OF LREAL;
END_VAR
END_METHOD

METHOD CALCULATECONFIGURATION : WORD
VAR_IN_OUT
	AXESGROUP : AXES_GROUP_KIN;
	ALRPOSFLANGE : ARRAY [1..6] OF LREAL;
	ALRPOSAXES : ARRAY [1..6] OF LREAL;
	AICONFIGURATION : ARRAY [1..6] OF INT;
END_VAR
END_METHOD

(* ---- L_MC4P_ITRAFOINTERFACE.itf ---- *)
INTERFACE L_MC4P_ITRAFOINTERFACE
END_INTERFACE

METHOD BWDACC : BOOL
VAR_INPUT
	ICOORDPROVIDER : REFERENCE TO L_MC4P_KinCoordProvider;
END_VAR
VAR_OUTPUT
	SCERROR : L_MC4P_ErrorStruct;
END_VAR
VAR_IN_OUT
	SCTRAFOINFO : L_MC4P_TrafoInfo;
END_VAR
END_METHOD

METHOD BWDPOS : BOOL
VAR_INPUT
	ICOORDPROVIDER : REFERENCE TO L_MC4P_KinCoordProvider;
END_VAR
VAR_OUTPUT
	SCERROR : L_MC4P_ErrorStruct;
END_VAR
VAR_IN_OUT
	SCTRAFOINFO : L_MC4P_TrafoInfo;
END_VAR
END_METHOD

METHOD BWDVEL : BOOL
VAR_INPUT
	ICOORDPROVIDER : REFERENCE TO L_MC4P_KinCoordProvider;
END_VAR
VAR_OUTPUT
	SCERROR : L_MC4P_ErrorStruct;
END_VAR
VAR_IN_OUT
	SCTRAFOINFO : L_MC4P_TrafoInfo;
END_VAR
END_METHOD

METHOD CALCPASSIVEJOINTS : L_IE1P_Error
VAR_INPUT
	PFLANGE_POS : POINTER TO ARRAY [1..6] OF LREAL;
	PJOINT_POS : POINTER TO ARRAY [1..6] OF LREAL;
	PPASSIVEJOINT_POS : POINTER TO ARRAY [1..6, 1..3] OF LREAL;
END_VAR
END_METHOD

METHOD CALCULATECONFIGURATION : L_IE1P_Error
VAR_INPUT
	PJOINT_POS : POINTER TO ARRAY [1..6] OF LREAL;
END_VAR
VAR_IN_OUT
	SCTRAFOINFO : L_MC4P_TrafoInfo;
END_VAR
END_METHOD

METHOD FWDACC : BOOL
VAR_INPUT
	ICOORDPROVIDER : REFERENCE TO L_MC4P_KinCoordProvider;
END_VAR
VAR_OUTPUT
	SCERROR : L_MC4P_ErrorStruct;
END_VAR
VAR_IN_OUT
	SCTRAFOINFO : L_MC4P_TrafoInfo;
END_VAR
END_METHOD

METHOD FWDPOS : BOOL
VAR_INPUT
	ICOORDPROVIDER : REFERENCE TO L_MC4P_KinCoordProvider;
END_VAR
VAR_OUTPUT
	SCERROR : L_MC4P_ErrorStruct;
END_VAR
VAR_IN_OUT
	SCTRAFOINFO : L_MC4P_TrafoInfo;
END_VAR
END_METHOD

METHOD FWDVEL : BOOL
VAR_INPUT
	ICOORDPROVIDER : REFERENCE TO L_MC4P_KinCoordProvider;
END_VAR
VAR_OUTPUT
	SCERROR : L_MC4P_ErrorStruct;
END_VAR
VAR_IN_OUT
	SCTRAFOINFO : L_MC4P_TrafoInfo;
END_VAR
END_METHOD

METHOD GETTRAFOEXTENSION1 : L_MC4P_ITrafoExtension
VAR_OUTPUT
	PFB : POINTER TO L_MC4P_TrafoExtensionBase;
END_VAR
END_METHOD

METHOD MCS_ORIENTATIONCHECK : L_IE1P_Error
VAR_IN_OUT
	ICOORDPROVIDER : L_MC4P_KinCoordProvider;
END_VAR
END_METHOD

METHOD SETTRAFOEXTENSION1
VAR_INPUT
	TRAFOEXTENSION : L_MC4P_ITrafoExtension;
	PFB : POINTER TO L_MC4P_TrafoExtensionBase;
END_VAR
END_METHOD

(* ---- L_MC4P_VISUINTERFACE.itf ---- *)
INTERFACE L_MC4P_VISUINTERFACE
END_INTERFACE

METHOD COMMONMAIN
END_METHOD

(* ---- MC_KIN_REF.itf ---- *)
INTERFACE MC_KIN_REF
END_INTERFACE

METHOD GETPARAITF : L_MC4P_IKinParamExtern
END_METHOD

METHOD GETTRAFOITF : L_MC4P_ITrafoExtern
END_METHOD

METHOD LINKEDAXESGROUP_GET : POINTER TO AXES_GROUP_KIN
END_METHOD

METHOD LINKEDAXESGROUP_SET
VAR_INPUT
	LINKEDAXESGROUP : POINTER TO AXES_GROUP_KIN;
END_VAR
END_METHOD

METHOD SETACSAXISTYPE
VAR_OUTPUT
	AEAXES : ARRAY [1..6] OF L_MC4P_AxisType := [L_MC4P_AxisType.unconnected, L_MC4P_AxisType.unconnected, L_MC4P_AxisType.unconnected, L_MC4P_AxisType.unconnected, L_MC4P_AxisType.unconnected, L_MC4P_AxisType.unconnected];
END_VAR
END_METHOD

METHOD SETINITIALVALUESOFCONSTANTMCSAXES
VAR_OUTPUT
	ALRMCSPOS : ARRAY [1..6] OF LREAL := [0.0, 0.0, 0.0, 0.0, 0.0, 0.0];
END_VAR
END_METHOD

METHOD SETMCSAXISTYPE
VAR_OUTPUT
	AEAXES : ARRAY [1..6] OF L_MC4P_AxisType := [L_MC4P_AxisType.unconnected, L_MC4P_AxisType.unconnected, L_MC4P_AxisType.unconnected, L_MC4P_AxisType.unconnected, L_MC4P_AxisType.unconnected, L_MC4P_AxisType.unconnected];
END_VAR
END_METHOD

(* ---- MC_PATH_REF.itf ---- *)
INTERFACE MC_PATH_REF
END_INTERFACE

METHOD GETID : __XWORD
END_METHOD

METHOD GETPATHDATA : ARRAY [1..30] OF POINTER TO L_MC4P_Parameter_MCMove
END_METHOD

METHOD GETPATHDATAACTIVE : BOOL
END_METHOD

METHOD GETSTATUS : DWORD
END_METHOD

METHOD SETABORT
END_METHOD

METHOD SETACTIVEMFUNCTION
VAR_INPUT
	WACTIVEMFUNCTION : WORD;
END_VAR
END_METHOD

METHOD SETMOVEPATHACTIVE
VAR_INPUT
	XMOVEPATHACTIVE : BOOL;
END_VAR
END_METHOD

METHOD SETPATHDATAACTIVE
VAR_INPUT
	XPATHDATAACTIVE : BOOL;
END_VAR
END_METHOD

(* ---- ABC2QUAT.pou ---- *)
FUNCTION ABC2QUAT
VAR_INPUT
	A_DEG : LREAL;
	B_DEG : LREAL;
	C_DEG : LREAL;
	EROTATIONCONVENTION : L_UMTP_RotationConvention;
END_VAR
VAR_IN_OUT
	QUAT : ARRAY [1..4] OF LREAL;
END_VAR
END_FUNCTION

(* ---- ABC2R.pou ---- *)
FUNCTION ABC2R
VAR_INPUT
	A_DEG : LREAL;
	B_DEG : LREAL;
	C_DEG : LREAL;
	EROTATIONCONVENTION : L_UMTP_RotationConvention;
END_VAR
VAR_IN_OUT
	ROTMAT : ARRAY [1..3, 1..3] OF LREAL;
END_VAR
END_FUNCTION

(* ---- ABC2R_RAD.pou ---- *)
FUNCTION ABC2R_RAD
VAR_INPUT
	A_RAD : LREAL;
	B_RAD : LREAL;
	C_RAD : LREAL;
	EROTATIONCONVENTION : L_UMTP_RotationConvention;
END_VAR
VAR_IN_OUT
	ROTMAT : ARRAY [1..3, 1..3] OF LREAL;
END_VAR
END_FUNCTION

(* ---- ACCKART2ZYL.pou ---- *)
FUNCTION ACCKART2ZYL
VAR_IN_OUT
	ALRINPOSZYL : ARRAY [1..6] OF LREAL;
	ALRINACCKART : ARRAY [1..6] OF LREAL;
	ALRT_10 : ARRAY [1..4, 1..4] OF LREAL;
	ALROUT : ARRAY [1..6] OF LREAL;
END_VAR
END_FUNCTION

(* ---- ACCZYL2KART.pou ---- *)
FUNCTION ACCZYL2KART
VAR_IN_OUT
	ALRINPOSZYL : ARRAY [1..6] OF LREAL;
	ALRINACCZYL : ARRAY [1..6] OF LREAL;
	ALRT_01 : ARRAY [1..4, 1..4] OF LREAL;
	ALROUT : ARRAY [1..6] OF LREAL;
END_VAR
END_FUNCTION

(* ---- CALCCIRCCENTER2D.pou ---- *)
FUNCTION CALCCIRCCENTER2D : BOOL
VAR_OUTPUT
	ALRCENTER : ARRAY [1..2] OF LREAL;
END_VAR
VAR_IN_OUT
	ALRX0 : ARRAY [1..2] OF LREAL;
	ALRX1 : ARRAY [1..2] OF LREAL;
	LRR : LREAL;
	PATHCHOICE : MC_CIRC_PATHCHOICE;
END_VAR
END_FUNCTION

(* ---- CALCQUATROTANGLE.pou ---- *)
FUNCTION CALCQUATROTANGLE : BOOL
VAR_INPUT
	PQUAT1 : POINTER TO ARRAY [1..4] OF LREAL;
	PQUAT2 : POINTER TO ARRAY [1..4] OF LREAL;
	PTHETA : POINTER TO LREAL;
END_VAR
END_FUNCTION

(* ---- CHECKQUATERNION.pou ---- *)
FUNCTION CHECKQUATERNION : BOOL
VAR_INPUT
	PQUAT : POINTER TO ARRAY [1..4] OF LREAL;
END_VAR
END_FUNCTION

(* ---- COORD2T.pou ---- *)
FUNCTION COORD2T
VAR_IN_OUT
	T : ARRAY [1..4, 1..4] OF LREAL;
	COORDTRANSFORM : MC_COORD_REF;
	EROTATIONCONVENTION : L_UMTP_RotationConvention;
END_VAR
END_FUNCTION

(* ---- COPYLISTELEMENTDATA.pou ---- *)
FUNCTION COPYLISTELEMENTDATA : BOOL
VAR_INPUT
	PDEST : POINTER TO L_MC4P_ListElement;
	PSOUR : POINTER TO L_MC4P_ListElement;
END_VAR
END_FUNCTION

(* ---- FAILED.pou ---- *)
FUNCTION FAILED : BOOL
VAR_INPUT
	SCERROR : REFERENCE TO L_MC4P_ErrorStruct;
END_VAR
END_FUNCTION

(* ---- FINDINTERVAL.pou ---- *)
FUNCTION FINDINTERVAL : BOOL
VAR_INPUT
	LRVALUE : LREAL;
	PLRVALUES : POINTER TO LREAL;
	NDATA : UDINT;
	XZEROBASED : BOOL;
	XTRYFIRST : BOOL;
END_VAR
VAR_IN_OUT
	UDIINTERVAL : UDINT;
END_VAR
END_FUNCTION

(* ---- GETBOOLEANPROPERTY.pou ---- *)
FUNCTION GETBOOLEANPROPERTY : BOOL
VAR_INPUT
	STKEY : WSTRING;
END_VAR
END_FUNCTION

(* ---- GETCOMPANY.pou ---- *)
FUNCTION GETCOMPANY : WSTRING
END_FUNCTION

(* ---- GETNUMBERPROPERTY.pou ---- *)
FUNCTION GETNUMBERPROPERTY : DINT
VAR_INPUT
	STKEY : WSTRING;
END_VAR
END_FUNCTION

(* ---- GETTEXTPROPERTY.pou ---- *)
FUNCTION GETTEXTPROPERTY : WSTRING
VAR_INPUT
	STKEY : WSTRING;
END_VAR
END_FUNCTION

(* ---- GETTEXTPROPERTY2.pou ---- *)
FUNCTION GETTEXTPROPERTY2 : POINTER TO WSTRING
VAR_INPUT
	STKEY : WSTRING;
END_VAR
END_FUNCTION

(* ---- GETTITLE.pou ---- *)
FUNCTION GETTITLE : WSTRING
END_FUNCTION

(* ---- GETVERSION.pou ---- *)
FUNCTION GETVERSION : VERSION
END_FUNCTION

(* ---- GETVERSIONPROPERTY.pou ---- *)
FUNCTION GETVERSIONPROPERTY : VERSION
VAR_INPUT
	STKEY : WSTRING;
END_VAR
END_FUNCTION

(* ---- INITELLIPTICALINTEGRALLUT.pou ---- *)
FUNCTION INITELLIPTICALINTEGRALLUT
END_FUNCTION

(* ---- INITELLIPTICALINTEGRALLUT_2.pou ---- *)
FUNCTION INITELLIPTICALINTEGRALLUT_2
END_FUNCTION

(* ---- L_MC4P_CHECK_PATHREFVALID.pou ---- *)
FUNCTION L_MC4P_CHECK_PATHREFVALID : BOOL
VAR_INPUT
	PATHREF : MC_PATH_REF;
END_VAR
END_FUNCTION

(* ---- L_MC4P_FORCELREAL.pou ---- *)
FUNCTION L_MC4P_FORCELREAL : BOOL
VAR_INPUT
	LRACTUAL : REFERENCE TO LREAL;
	LRWANTED : LREAL;
END_VAR
END_FUNCTION

(* ---- L_MC4P_GETPATHDYN.pou ---- *)
FUNCTION L_MC4P_GETPATHDYN
VAR_INPUT
	PV : POINTER TO LREAL;
	PA : POINTER TO LREAL;
END_VAR
VAR_OUTPUT
	VEL_PATH : LREAL;
	ACC_PATH : LREAL;
END_VAR
END_FUNCTION

(* ---- LISTELEMENTISCARTESIAN.pou ---- *)
FUNCTION LISTELEMENTISCARTESIAN : BOOL
VAR_INPUT
	PLISTELEMENT : POINTER TO L_MC4P_ListElement;
END_VAR
END_FUNCTION

(* ---- MOVEELLIPTICAL_ANGLE2PARAM.pou ---- *)
FUNCTION MOVEELLIPTICAL_ANGLE2PARAM : LREAL
VAR_INPUT
	LRANGLE : LREAL;
	LRA : LREAL;
	LRB : LREAL;
END_VAR
END_FUNCTION

(* ---- MOVEELLIPTICAL_CALCELLIPTICINTEGRAL.pou ---- *)
FUNCTION MOVEELLIPTICAL_CALCELLIPTICINTEGRAL : LREAL
VAR_INPUT
	E : LREAL;
	T : LREAL;
END_VAR
END_FUNCTION

(* ---- MOVEELLIPTICAL_PARAM2ANGLE.pou ---- *)
FUNCTION MOVEELLIPTICAL_PARAM2ANGLE : LREAL
VAR_INPUT
	LRPARAM : LREAL;
	LRA : LREAL;
	LRB : LREAL;
END_VAR
END_FUNCTION

(* ---- QUAT2ABC.pou ---- *)
FUNCTION QUAT2ABC
VAR_INPUT
	EROTATIONCONVENTION : L_UMTP_RotationConvention;
	XCALCABC2 : BOOL := TRUE;
END_VAR
VAR_IN_OUT
	ABC : ARRAY [1..3] OF LREAL;
	ABC2 : ARRAY [1..3] OF LREAL;
	QUAT : ARRAY [1..4] OF LREAL;
END_VAR
END_FUNCTION

(* ---- QUAT2ABC_EXTENDED.pou ---- *)
FUNCTION QUAT2ABC_EXTENDED : L_MC4P_ErrorStruct
VAR_INPUT
	EROTATIONCONVENTION : L_UMTP_RotationConvention;
	ALREXPECTEDABC : ARRAY [1..3] OF LREAL;
	AXROTANGLESFIXED : ARRAY [1..3] OF BOOL;
END_VAR
VAR_IN_OUT
	ABC : ARRAY [1..3] OF LREAL;
	QUAT : ARRAY [1..4] OF LREAL;
END_VAR
END_FUNCTION

(* ---- QUAT2R.pou ---- *)
FUNCTION QUAT2R
VAR_IN_OUT
	ROTMAT : ARRAY [1..3, 1..3] OF LREAL;
	QUAT : ARRAY [1..4] OF LREAL;
END_VAR
END_FUNCTION

(* ---- R2ABC.pou ---- *)
FUNCTION R2ABC
VAR_INPUT
	EROTATIONCONVENTION : L_UMTP_RotationConvention;
	XCALCABC2 : BOOL := TRUE;
END_VAR
VAR_IN_OUT
	ABC : ARRAY [1..3] OF LREAL;
	ABC2 : ARRAY [1..3] OF LREAL;
	ROTMAT : ARRAY [1..3, 1..3] OF LREAL;
END_VAR
END_FUNCTION

(* ---- R2ABC_EXTENDED.pou ---- *)
FUNCTION R2ABC_EXTENDED : L_MC4P_ErrorStruct
VAR_INPUT
	EROTATIONCONVENTION : L_UMTP_RotationConvention;
	ALREXPECTEDABC : ARRAY [1..3] OF LREAL;
	AXROTANGLESFIXED : ARRAY [1..3] OF BOOL;
END_VAR
VAR_IN_OUT
	ABC : ARRAY [1..3] OF LREAL;
	ROTMAT : ARRAY [1..3, 1..3] OF LREAL;
END_VAR
END_FUNCTION

(* ---- R2OMEGA.pou ---- *)
FUNCTION R2OMEGA : ARRAY [1..3] OF LREAL
VAR_INPUT
	LRFCYCLE : LREAL;
END_VAR
VAR_IN_OUT
	ALRROLD : ARRAY [1..3, 1..3] OF LREAL;
	ALRRNEW : ARRAY [1..3, 1..3] OF LREAL;
END_VAR
END_FUNCTION

(* ---- R2QUAT.pou ---- *)
FUNCTION R2QUAT
VAR_IN_OUT
	QUAT : ARRAY [1..4] OF LREAL;
	ROTMAT : ARRAY [1..3, 1..3] OF LREAL;
END_VAR
END_FUNCTION

(* ---- STRETCHPROFILETOTIME_RAST2RAST.pou ---- *)
FUNCTION STRETCHPROFILETOTIME_RAST2RAST
VAR_INPUT
	LRTDESIRED : LREAL;
	LRTASKCYCLE : LREAL;
END_VAR
VAR_IN_OUT
	SCPROFILEDATA : L_MC1P_ProfileData;
	SCPARAM : L_MC1P_ProfileParameter;
END_VAR
END_FUNCTION

(* ---- SUCCEEDED.pou ---- *)
FUNCTION SUCCEEDED : BOOL
VAR_INPUT
	SCERROR : REFERENCE TO L_MC4P_ErrorStruct;
END_VAR
END_FUNCTION

(* ---- T2COORD.pou ---- *)
FUNCTION T2COORD
VAR_INPUT
	EROTATIONCONVENTION : L_UMTP_RotationConvention;
END_VAR
VAR_IN_OUT
	COORDREF : MC_COORD_REF;
	T_01 : ARRAY [1..4, 1..4] OF LREAL;
END_VAR
END_FUNCTION

(* ---- T2COORD_EXTENDED.pou ---- *)
FUNCTION T2COORD_EXTENDED : L_MC4P_ErrorStruct
VAR_INPUT
	EROTATIONCONVENTION : L_UMTP_RotationConvention;
	ALREXPECTEDABC : ARRAY [1..3] OF LREAL;
	AXROTANGLESFIXED : ARRAY [1..3] OF BOOL;
END_VAR
VAR_IN_OUT
	COORDREF : MC_COORD_REF;
	T_01 : ARRAY [1..4, 1..4] OF LREAL;
END_VAR
END_FUNCTION

(* ---- T2COORD_EXTENDED_FRAME.pou ---- *)
FUNCTION T2COORD_EXTENDED_FRAME : L_MC4P_ErrorStruct
VAR_INPUT
	EROTATIONCONVENTION : L_UMTP_RotationConvention;
	ALREXPECTEDABC : ARRAY [1..3] OF LREAL;
	AXROTANGLESFIXED : ARRAY [1..3] OF BOOL;
END_VAR
VAR_IN_OUT
	COORDREF : MC_COORD_REF;
	T_01 : L_UMTP_RobotPos;
END_VAR
END_FUNCTION

(* ---- T2R.pou ---- *)
FUNCTION T2R
VAR_IN_OUT
	ROTMAT : ARRAY [1..3, 1..3] OF LREAL;
	T : ARRAY [1..4, 1..4] OF LREAL;
END_VAR
END_FUNCTION

(* ---- VELKART2ZYL.pou ---- *)
FUNCTION VELKART2ZYL
VAR_IN_OUT
	ALRINPOSZYL : ARRAY [1..6] OF LREAL;
	ALRINVELKART : ARRAY [1..6] OF LREAL;
	ALRT_10 : ARRAY [1..4, 1..4] OF LREAL;
	ALROUT : ARRAY [1..6] OF LREAL;
END_VAR
END_FUNCTION

(* ---- VELZYL2KART.pou ---- *)
FUNCTION VELZYL2KART
VAR_IN_OUT
	ALRINPOSZYL : ARRAY [1..6] OF LREAL;
	ALRINVELZYL : ARRAY [1..6] OF LREAL;
	ALRT_01 : ARRAY [1..4, 1..4] OF LREAL;
	ALROUT : ARRAY [1..6] OF LREAL;
END_VAR
END_FUNCTION

(* ---- AXES_GROUP_BASE.pou ---- *)
FUNCTION_BLOCK AXES_GROUP_BASE EXTENDS IoDrvBase
VAR
	M_PAXISCONNECTOR : POINTER TO IoConfigConnector;
	M_IIODRV : ICmpIoDrv;
	M_IIODRVPARAMETER : ICmpIoDrvParameter;
	DWIODRVDEVICEID : DWORD;
	WIODRVDEVICETYPE : WORD;
END_VAR
END_FUNCTION_BLOCK
